// TIA Portal V18 program export: 6 tag tables, 0 data types, 2 data blocks, 13 code blocks (in call order from the OBs), 43 instance data blocks

VAR_GLOBAL   // PLC tag table "Alarms"
   "Alarm Main 1/5" AT %MW600 : Word;
   "Alarm Main 2/5" AT %MW602 : Word;
   "Alarm Main 3/5" AT %MW604 : Word;
   "Alarm Main 4/5" AT %MW606 : Word;
   "Alarm Main 5/5" AT %MW608 : Word;
   "Alarm Main 6" AT %MW610 : Word;
   "Alarm Main 7" AT %MW612 : Word;
   "AL-Drive Left Slow Limit Angle" AT %M600.0 : Bool;
   "AL-Drive Left Stop Limit LS" AT %M600.1 : Bool;
   "AL-Drive Left Stop Limit Angle" AT %M600.2 : Bool;
   "AL-Drive Left Stop Limit" AT %M600.3 : Bool;
   "AL-Drive Right Slow Limit Angle" AT %M600.4 : Bool;
   "AL-Drive Right Stop Limit LS" AT %M600.5 : Bool;
   "AL-Drive Right Stop Limit Angle" AT %M600.6 : Bool;
   "AL-Drive Right Stop Limit" AT %M600.7 : Bool;
   "AL-Rotunda Left Slow Limit" AT %M601.0 : Bool;
   "AL-Rotunda Right Slow Limit" AT %M601.1 : Bool;
   "AL-Rotunda Slow Limit" AT %M601.2 : Bool;
   "AL-Rotunda Left Stop Limit LS" AT %M601.3 : Bool;
   "AL-Rotunda Left FW Stop Limit" AT %M601.4 : Bool;
   "AL-Rotunda Left BW Stop Limit" AT %M601.5 : Bool;
   "AL-Rotunda Right Stop Limit LS" AT %M601.6 : Bool;
   "AL-Rotunda Right FW Stop Limit" AT %M601.7 : Bool;
   "AL-Rotunda Right BW Stop Limit" AT %M602.0 : Bool;
   "AL-Rotunda FW Stop Limit All" AT %M602.1 : Bool;
   "AL-Rotunda BW Stop Limit All" AT %M602.2 : Bool;
   "AL-Tunnel FW Slow Limit Laser" AT %M602.3 : Bool;
   "AL-Tunnel FW Slow Limit LS" AT %M602.4 : Bool;
   "AL-Tunnel FW Slow Limit PhotoCell" AT %M602.5 : Bool;
   "AL-Tunnel FW Slow Limit UltraSonic" AT %M602.6 : Bool;
   "AL-Tunnel FW Slow Limit All" AT %M602.7 : Bool;
   "AL-Tunnel BW Slow Limit Laser" AT %M603.0 : Bool;
   "AL-Tunnel BW Slow Limit LS" AT %M603.1 : Bool;
   "AL-Tunnel BW Slow Limit All" AT %M603.2 : Bool;
   "AL-Tunnel FW Stop Limit Laser" AT %M603.3 : Bool;
   "AL-Tunnel FW Stop Limit LS" AT %M603.4 : Bool;
   "AL-Tunnel FW Stop Limit PhotoCell Left" AT %M603.5 : Bool;
   "AL-Tunnel FW Stop Limit PhotoCell Mid" AT %M603.6 : Bool;
   "AL-Tunnel FW Stop Limit PhotoCell Right" AT %M603.7 : Bool;
   "AL-Tunnel FW Stop Limit All" AT %M604.0 : Bool;
   "AL-Tunnel FW Emergency Stop Limit" AT %M604.1 : Bool;
   "AL-Tunnel BW Stop Limit Laser" AT %M604.2 : Bool;
   "AL-Tunnel BW Stop Limit LS" AT %M604.3 : Bool;
   "AL-Tunnel BW Stop Limit All" AT %M604.4 : Bool;
   "AL-Tunnel BW Emergency Stop Limit" AT %M604.5 : Bool;
   "AL-Slow Activated" AT %M604.6 : Bool;
   "AL-Drive Slow Limit All" AT %M604.7 : Bool;
   "AL-Tunnel FW Slow Limit Slope" AT %M605.0 : Bool;
   "AL-Tunnel FW Stop Limit Slope" AT %M605.1 : Bool;
   "AL-Tunnel BW Slow Limit Slope" AT %M605.2 : Bool;
   "AL-Tunnel BW Stop Limit Slope" AT %M605.3 : Bool;
   "AL-Drivers Fault, Wheel" AT %M605.4 : Bool;
   "AL-Wheel Fuse" AT %M605.5 : Bool;
   "AL-Up Stop Limit, Wire" AT %M605.6 : Bool;
   "AL-Up Stop Limit, Max Slope" AT %M605.7 : Bool;
   "AL-Up Stop Limit, BW LS" AT %M606.0 : Bool;
   "AL-Up Stop Limit, All" AT %M606.1 : Bool;
   "AL-Down Stop Limit, Wire" AT %M606.2 : Bool;
   "AL-Down Stop Limit, Object" AT %M606.3 : Bool;
   "AL-Down Stop Limit, Min Slope" AT %M606.4 : Bool;
   "AL-Down Stop Limit, FW LS" AT %M606.5 : Bool;
   "AL-Down Stop Limit, All" AT %M606.6 : Bool;
   "AL-SafetyShoe Activated" AT %M606.7 : Bool;
   "AL-SafetyShoe Cable Problem" AT %M607.0 : Bool;
   "AL-AutoLeveller Up Over Work" AT %M607.1 : Bool;
   "AL-AutoLeveller Down Over Work" AT %M607.2 : Bool;
   "AL-AutoLeveller Touch" AT %M607.3 : Bool;
   "AL-Hydraulic Motor MKS" AT %M607.4 : Bool;
   "AL-Up Button Pressed" AT %M607.5 : Bool;
   "AL-Down Button Pressed" AT %M607.6 : Bool;
   "AL-AutoLeveller Motor Fault" AT %M607.7 : Bool;
   "AL-Left Canopy Touch" AT %M608.0 : Bool;
   "AL-Right Canopy Touch" AT %M608.1 : Bool;
   "AL-Left Canopy MKS" AT %M608.2 : Bool;
   "AL-Right Canopy MKS" AT %M608.3 : Bool;
   "AL-Canopy FW Button Pressed" AT %M608.4 : Bool;
   "AL-Canopy BW Button Pressed" AT %M608.5 : Bool;
   "AL-Cab Left Stop Limit, LS" AT %M608.6 : Bool;
   "AL-Cab Left Stop Limit, Angle" AT %M608.7 : Bool;
   "AL-Cab Left Stop Limit, All" AT %M609.0 : Bool;
   "AL-Cab Right Stop Limit, LS" AT %M609.1 : Bool;
   "AL-Cab Right Stop Limit, Angle" AT %M609.2 : Bool;
   "AL-Cab Right Stop Limit, All" AT %M609.3 : Bool;
   "AL-Driver Fault, Cab" AT %M609.4 : Bool;
   "AL-Cab Motor MKS" AT %M609.5 : Bool;
   "AL-Cab Left Button Pressed" AT %M609.6 : Bool;
   "AL-Cab Right Button Pressed" AT %M609.7 : Bool;
   "AL-Cab Floor FW Button Pressed" AT %M610.0 : Bool;
   "AL-Cab Floor BW Button Pressed" AT %M610.1 : Bool;
   "AL-Cab Floor Motor Fault" AT %M610.2 : Bool;
   "AL-PBB in Off Mode" AT %M610.3 : Bool;
   "AL-PBB in Auto Mode" AT %M610.4 : Bool;
   "AL-Left Emergency Stop Pressed" AT %M610.5 : Bool;
   "AL-Right Emergency Stop Pressed" AT %M610.6 : Bool;
   "AL-CP Emergency Stop Pressed" AT %M610.7 : Bool;
   "AL-Emergency Stop Pressed" AT %M611.0 : Bool;
   "AL-ByPass Activated" AT %M611.1 : Bool;
   "AL-PBB in On Mode" AT %M611.2 : Bool;
   "AL-Main Contactor ON" AT %M611.3 : Bool;
   "AL-FAULT" AT %M611.4 : Bool;
   "AL-SafetyBarrier Activated" AT %M611.5 : Bool;
   "AL-No Electricity" AT %M611.6 : Bool;
   "AL-Service-Hose" AT %M619.0 : Bool;
   "AL-Service-GPU" AT %M619.1 : Bool;
   "AL-Service-PCA" AT %M619.2 : Bool;
   "AL-Service" AT %M619.3 : Bool;
   "AL-Drive Angle LS FW Stop" AT %M619.5 : Bool;
   "AL-Drive Angle LS BW Stop" AT %M619.4 : Bool;
   "AL-PBB HOME" AT %M619.6 : Bool;
   "AL-AutoLeveller Down" AT %M614.0 : Bool;
   "AL-AutoLeveller Up" AT %M614.1 : Bool;
END_VAR

VAR_GLOBAL   // PLC tag table "Analog_Clock"
   "Rotunda Angle input" AT %IW160 : Int;
   "Drive Angle input" AT %IW164 : Int;
   "Cabin Angle input" AT %IW166 : Int;
   "WireDraw Encoder input" AT %IW176 : Int;
   "Laser input" AT %IW162 : Int;
   "Left Driver Analog input" AT %QW160 : Int;
   "Right Driver Analog input" AT %QW162 : Int;
   "Cab Driver Analog input" AT %QW176 : Int;
   "Slow Mode input" AT %M226.1 : Bool;
   "Canopy Touch Memo" AT %M217.4 : Bool;
END_VAR

VAR_GLOBAL   // PLC tag table "HMI"
   "HMI SafetyEdge Bypass" AT %M800.0 : Bool;
   "HMI R1 - Plane Door Light" AT %M800.1 : Bool;
   "HMI R2 - Plane Door Light" AT %M800.2 : Bool;
   "HMI R3 - Drive Unit Light" AT %M800.3 : Bool;
   "HMI R4 - Cabin Front Light" AT %M800.4 : Bool;
   "HMI R6 - SafetyEdge Light" AT %M800.5 : Bool;
   "HMI - Lamp Test Button" AT %M800.6 : Bool;
   "HMI - Floor Auto Mode" AT %M800.7 : Bool;
   "HMI - AntiCrash UltraSonic ByPass" AT %M801.0 : Bool;
   "HMI - Int Light Button" AT %M801.1 : Bool;
   "HMI - Fire Siren Acitve/Passive" AT %M801.2 : Bool;
   "HMI - Auto Floor" AT %M801.3 : Bool;
END_VAR

VAR_GLOBAL   // PLC tag table "Inputs"
   "Driver Alarm Left" AT %I0.0 : Bool;
   "Driver Fault Left" AT %I0.1 : Bool;
   "Driver Alarm Right" AT %I0.2 : Bool;
   "Driver Fault Right" AT %I0.3 : Bool;
   "Cab Driver Fault" AT %I0.5 : Bool;
   "Drive LSW Stop Left" AT %I2.0 : Bool;
   "Drive LSW Stop Right" AT %I2.1 : Bool;
   SafetyEdge AT %I2.4 : Bool;
   "Em Stop Left" AT %I2.2 : Bool;
   "Em Stop Right" AT %I2.3 : Bool;
   "Canopy Touch Left" AT %I2.7 : Bool;
   "Canopy Touch Right" AT %I3.0 : Bool;
   "Bumper Touch Left" AT %I3.1 : Bool;
   "Bumper Touch Mid" AT %I3.2 : Bool;
   "Bumper Touch Right" AT %I3.3 : Bool;
   "PhotoCell for AirCraft" AT %I3.4 : Bool;
   "UltraSonic for AirCraft" AT %I3.5 : Bool;
   "UltraSonic for Object" AT %I3.6 : Bool;
   "AutoLeveller Touch" AT %I3.7 : Bool;
   "AutoLeveller Up Sensor" AT %I4.0 : Bool;
   "AutoLeveller Down Sensor" AT %I4.1 : Bool;
   "Cabin LSW Left" AT %I4.4 : Bool;
   "Cabin LSW Right" AT %I4.5 : Bool;
   "PCA Active" AT %I15.5 : Bool;
   "Rotunda LSW Left Stop" AT %I4.6 : Bool;
   "Rotunda LSW Right Stop" AT %I4.7 : Bool;
   "Tunnel LSW FW Slow İnput" AT %I5.2 : Bool;   // FW Slow
   "Tunnel LSW BW Slow İnput" AT %I5.3 : Bool;   // BW Slow
   "Tunnel LSW FW Stop İnput" AT %I5.4 : Bool;   // FW Stop
   "Tunnel LSW BW Stop İnput" AT %I5.5 : Bool;   // BW Stop
   "Tunnel LSW FW Em Stop İnput" AT %I5.6 : Bool;   // FW Em Stop
   "Tunnel LSW BW Em Stop İnput" AT %I5.7 : Bool;   // BW Em Stop
   "Rotunda Fire Detector" AT %I6.0 : Bool;
   "Drive Wheel Fuse" AT %I6.7 : Bool;
   "Fuse Hydraulic" AT %I6.1 : Bool;
   "Fuse Cab" AT %I6.2 : Bool;
   "Phase Relay - PCR" AT %I7.0 : Bool;
   "SafetyShoe-1" AT %I10.0 : Bool;
   "SafetyShoe-2" AT %I10.1 : Bool;
   "Fuse Left Canopy" AT %I10.3 : Bool;
   "Fuse Right Canopy" AT %I10.4 : Bool;
   "Fuse Cab Floor" AT %I10.2 : Bool;
   "Fuse AutoLeveller" AT %I10.5 : Bool;
   "Button ByPass" AT %I11.0 : Bool;
   "Button Reset" AT %I11.1 : Bool;
   "Button Light Int" AT %I11.2 : Bool;
   "Button Ext Light" AT %I11.3 : Bool;
   "Button BackUp" AT %I11.4 : Bool;
   "Em Stop Button" AT %I11.5 : Bool;
   "Key-1 ON" AT %I11.7 : Bool;
   "Key-2 OFF" AT %I11.6 : Bool;
   "Cab Button Left" AT %I12.0 : Bool;
   "Cab Button Right" AT %I12.1 : Bool;
   "Button PBB Up" AT %I12.2 : Bool;
   "Button Pbb Down" AT %I12.3 : Bool;
   "Canopy Button BW" AT %I12.5 : Bool;
   "Canopy Button FW" AT %I12.4 : Bool;
   "Cab Floor FW" AT %I12.6 : Bool;
   "Cab Floor BW" AT %I12.7 : Bool;
   "JoyStick X22 L2" AT %I13.0 : Bool;
   "JoyStick X33 FW" AT %I13.1 : Bool;
   "JoyStick X44 L3" AT %I13.2 : Bool;
   "JoyStick X55 BW" AT %I13.3 : Bool;
   "JoyStick Y22 L2" AT %I13.4 : Bool;
   "JoyStick Y33 RGHT" AT %I13.5 : Bool;
   "JoyStick Y44 L3" AT %I13.6 : Bool;
   "JoyStick Y55 LFT" AT %I13.7 : Bool;
   "JoyStick 91 Brake" AT %I14.0 : Bool;
   "Fuse 1Power Supply" AT %I6.3 : Bool;
   "Fuse 2Power Supply" AT %I6.4 : Bool;
   "Fuse Phase Control Relay" AT %I6.5 : Bool;
   "GPU2 Active" AT %I15.3 : Bool;
   "Fire Detector Cabin" AT %I4.3 : Bool;
   "Fuse Hose Ritriver" AT %I6.6 : Bool;
   Fuse AT %I7.5 : Bool;
   "PCA Error" AT %I15.6 : Bool;
   "GPU2 Error" AT %I15.4 : Bool;
   "GPU1 Active" AT %I15.1 : Bool;
   "GPU1 Error" AT %I15.2 : Bool;
   "Hose Active" AT %I15.7 : Bool;
END_VAR

VAR_GLOBAL   // PLC tag table "MemoryType"
   "PBB Off Mode" AT %M200.0 : Bool;
   "PBB On Mode" AT %M200.1 : Bool;
   "PBB Auto Mode" AT %M200.2 : Bool;
   "Emergency Stop Button Pressed" AT %M200.3 : Bool;
   "Tunnel FW Em Stop LS M" AT %M200.4 : Bool;
   "Tunnel BW Em Stop LS M" AT %M200.5 : Bool;
   "Start M" AT %M200.6 : Bool;
   "Fuse Problem Major" AT %M200.7 : Bool;
   "AutoLeveller Fault" AT %M201.0 : Bool;
   "AutoLeveller Up Over Work" AT %M201.1 : Bool;
   "AutoLeveller Down Over Work" AT %M201.2 : Bool;
   "Driver Error Left" AT %M201.3 : Bool;
   "Driver Error Right" AT %M201.4 : Bool;
   "Wheel Drivers Fault" AT %M201.5 : Bool;
   "SafetyShoe Siren&Info" AT %M201.6 : Bool;
   "SafetyBarrier Activated" AT %M201.7 : Bool;
   "Fault Occurred Major" AT %M202.1 : Bool;
   "Cabin Motor Driver Fault" AT %M202.2 : Bool;
   "Fault Occured Minor" AT %M202.3 : Bool;
   OK AT %M202.4 : Bool;
   "FW L1" AT %M202.5 : Bool;
   "FW L2" AT %M202.6 : Bool;
   "FW L3" AT %M202.7 : Bool;
   "BW L1" AT %M203.0 : Bool;
   "BW L2" AT %M203.1 : Bool;
   "BW L3" AT %M203.2 : Bool;
   "LFT L1" AT %M203.3 : Bool;
   "LFT L2" AT %M203.4 : Bool;
   "LFT L3" AT %M203.5 : Bool;
   "RGHT L1" AT %M203.6 : Bool;
   "RGHT L2" AT %M203.7 : Bool;
   "RGHT L3" AT %M204.0 : Bool;
   "JS Mid M" AT %M204.1 : Bool;
   "SafetyShoe Activated" AT %M204.2 : Bool;
   "AutoLeveller Up" AT %M204.3 : Bool;
   "AutoLeveller Down" AT %M204.4 : Bool;
   "sanal kesici (1)" AT %M204.5 : Bool;
   "Down Stop Object Limit" AT %M204.6 : Bool;
   "SafetyShoe Long Press" AT %M204.7 : Bool;
   "SS Cable Problem" AT %M205.0 : Bool;
   "AutoSafety Cross" AT %M205.1 : Bool;
   "AutoLeveller FW" AT %M205.2 : Bool;
   "AutoLeveller BW" AT %M205.3 : Bool;
   "Autoleveler temp count" AT %M205.4 : Bool;
   "Fuse Problem Minor" AT %M205.7 : Bool;
   "Wire Up Stop PBB" AT %M206.0 : Bool;
   "Slope Stop Up" AT %M206.1 : Bool;
   "Wire Up Stop PBB Limit All" AT %M206.2 : Bool;
   "Wire Down Stop PBB" AT %M206.3 : Bool;
   "Slope Stop Down" AT %M206.4 : Bool;
   "Down Stop Object" AT %M206.5 : Bool;
   "Down Stop PBB All" AT %M206.6 : Bool;
   "Speed L1" AT %IW100 : Int;
   "Speed L2" AT %IW102 : Int;
   "Speed L3" AT %IW104 : Int;
   "Slow Activated" AT %M207.2 : Bool;
   "Drive Slow Limit All" AT %M207.3 : Bool;
   "FW Slow Limit All" AT %M207.4 : Bool;
   "BW Slow Limit All" AT %M207.5 : Bool;
   "FW M" AT %M207.6 : Bool;
   "BW M" AT %M207.7 : Bool;
   "FW-LFT" AT %M208.0 : Bool;
   "FW-RGHT" AT %M208.1 : Bool;
   "BW-LFT" AT %M208.2 : Bool;
   "BW-RGHT" AT %M208.3 : Bool;
   "Cross M" AT %M208.4 : Bool;
   "FW Stop All" AT %M208.5 : Bool;
   "BW Stop All" AT %M208.6 : Bool;
   "LFT Stop All" AT %M208.7 : Bool;
   "RGHT Stop All" AT %M209.0 : Bool;
   "FW Allowed" AT %M209.1 : Bool;
   "BW Allowed" AT %M209.2 : Bool;
   "LFT Allowed" AT %M209.3 : Bool;
   "RGHT Allowed" AT %M209.4 : Bool;
   "FW-LFT Allowed" AT %M209.5 : Bool;
   "FW-RGHT Allowed" AT %M209.6 : Bool;
   "BW-LFT Allowed" AT %M209.7 : Bool;
   "BW-RGHT Allowed" AT %M210.0 : Bool;
   "Drive Angle Stop Left" AT %M210.1 : Bool;
   "Drive LSW Left Stop" AT %M210.2 : Bool;
   "Drive Angle Stop Right" AT %M210.3 : Bool;
   "Drive LSW Right Stop" AT %M210.4 : Bool;
   "Drive Slow Left Limit" AT %M210.5 : Bool;
   "Drive Slow Right Limit" AT %M210.6 : Bool;
   "Rotunda FW Stop LFT" AT %M210.7 : Bool;
   "Brake Off Time" AT %ID106 : Time;
   "Rotunda BW Stop LFT" AT %M211.0 : Bool;
   "Rotunda FW Stop RGHT" AT %M211.1 : Bool;
   "Rotunda BW Stop RGHT" AT %M211.2 : Bool;
   "Rotunda FW Stop All" AT %M211.3 : Bool;
   "Rotunda BW Stop All" AT %M211.4 : Bool;
   "Tunnel Laser FW Slow Limit" AT %M211.5 : Bool;
   "Tunnel LSW FW Slow" AT %M211.6 : Bool;
   "PhotoCell Slow Limit" AT %M211.7 : Bool;
   "UltraSonic Slow Limit" AT %M212.0 : Bool;
   "AirCraft Seen Anime" AT %M212.1 : Bool;
   "Laser BW Slow Limit" AT %M212.2 : Bool;
   "LS BW Slow Limit" AT %M212.3 : Bool;
   "Laser FW Stop Limit" AT %M212.5 : Bool;
   "LS FW Stop Limit" AT %M212.7 : Bool;
   "Touch LFT Stop Limit" AT %M213.0 : Bool;
   "Touch Mid Stop Limit" AT %M213.1 : Bool;
   "Touch RGTH Stop Limit" AT %M213.2 : Bool;
   "AirCraft Touch Anime" AT %M213.3 : Bool;
   "Laser BW Stop Limit" AT %M213.4 : Bool;
   "LS BW Stop Limit" AT %M213.5 : Bool;
   "FW G120C Stop" AT %M213.7 : Bool;
   "BW G120C Stop" AT %M214.0 : Bool;
   "LFT G120C Stop" AT %M214.1 : Bool;
   "Right G120C Stop" AT %M214.2 : Bool;
   "FW-LFT G120C Stop" AT %M214.3 : Bool;
   "FW-RGHT G120C Stop" AT %M214.4 : Bool;
   "BW-LFT G120C Stop" AT %M214.5 : Bool;
   "BW-RGHT G120C Stop" AT %M214.6 : Bool;
   "Cab Angle Left Stop" AT %M214.7 : Bool;
   "Cab LS Left Stop" AT %M215.0 : Bool;
   "Cab Stop Left All" AT %M215.1 : Bool;
   "Cab Angle Right Stop" AT %M215.2 : Bool;
   "Cab LS Right Stop" AT %M215.3 : Bool;
   "Cab Stop Right All" AT %M215.4 : Bool;
   "Rotunda Stop Angle Rght" AT %M215.5 : Bool;
   "Rotunda Stop Angle LFT" AT %M215.6 : Bool;
   "Canopy BW Auto" AT %M216.0 : Bool;
   "canopy ok1" AT %M216.1 : Bool;
   "canopy ok2" AT %M216.2 : Bool;
   memo2 AT %M216.3 : Bool;
   memo AT %M216.4 : Bool;
   memo3 AT %M216.5 : Bool;
   memo4 AT %M220.0 : Bool;
   "SE ByPass" AT %M220.2 : Bool;
   "Tunnel Real Meter" AT %MD300 : Real;
   "Drive Angle Real Meter" AT %MD304 : Real;
   "Rotunda Angle Real Meter" AT %MD312 : Real;
   "Height Real" AT %MD332 : Real;
   "Cab Angle Real Meter" AT %MD348 : Real;
   "Rotunda Stop LS LFT" AT %M216.6 : Bool;
   "Rotunda Stop LS Rght" AT %M225.5 : Bool;
   "Slope Angel" AT %MD615 : Real;
   "Slope Vertical" AT %MD620 : Real;
   "Slope Stop All" AT %M225.6 : Bool;
   "Speed Active L1" AT %M225.7 : Bool;
   "Speed Active L2" AT %M226.2 : Bool;
   "Speed Active L3" AT %M226.3 : Bool;
   "Rotunda Slow Angle Rght" AT %M215.7 : Bool;
   "Rotunda Slow Angle LFT" AT %M216.7 : Bool;
   "Rotunda Slow Angle ALL" AT %M217.6 : Bool;
   "Slope Slow Down" AT %M206.7 : Bool;
   "Slope Slow Up" AT %M207.0 : Bool;
   "Slope Slow ALL" AT %M207.1 : Bool;
   "Fast Mode" AT %M226.0 : Bool;
   "Service GPU Active" AT %M202.0 : Bool;
   "Service PCA Active" AT %M205.5 : Bool;
   "Service Hose Active" AT %M205.6 : Bool;
   "Service Air Active" AT %M212.4 : Bool;
   "Drive Angle LS FW Stop" AT %M212.6 : Bool;
   "Drive Angle LS BW Stop" AT %M213.6 : Bool;
   "R6 - Cab Warning Light & Buzzer Test" AT %M226.4 : Bool;
END_VAR

VAR_GLOBAL   // PLC tag table "Outputs"
   "Left Driver On/Off" AT %Q0.0 : Bool;
   "Left Driver Reversing" AT %Q0.1 : Bool;
   "Left Driver Fault" AT %Q0.2 : Bool;
   "Left Driver DI4 STO" AT %Q0.3 : Bool;
   "Left Driver DI5 STO" AT %Q0.4 : Bool;
   "Right Driver On/Off" AT %Q0.5 : Bool;
   "Right Driver Reversing" AT %Q0.6 : Bool;
   "Right Driver Fault" AT %Q0.7 : Bool;
   "Right Driver DI4 STO" AT %Q1.0 : Bool;
   "Right Driver DI5 STO" AT %Q1.1 : Bool;
   "Cab Driver On/Off" AT %Q2.0 : Bool;
   "Cab Driver Reversing" AT %Q2.1 : Bool;
   "Cab Driver Fault Reset" AT %Q2.2 : Bool;
   "Cab Driver DI4 STO" AT %Q2.3 : Bool;
   "Cab Driver DI5 STO" AT %Q2.4 : Bool;
   "MC - Main Contactor" AT %Q3.0 : Bool;
   "C1 - Hydraulic" AT %Q3.1 : Bool;   // MC-105, MC-106, MC-107, MC-108, Cable No:200, MKS2
   "C2 - Hose power" AT %Q3.2 : Bool;
   "C3 - Tunnel Lights" AT %Q3.3 : Bool;
   "C4 - Tunnel Lights UPS" AT %Q3.4 : Bool;
   "C5 - Ext Lighting" AT %Q3.5 : Bool;
   "R2 - Bumper Red Light iptal" AT %Q3.7 : Bool;
   "R1 - SafetyEdge Red Light" AT %Q3.6 : Bool;   // MC-256 MC-257 MC-258, Cable No:204, F11
   "R4 - Mania Lights" AT %Q4.1 : Bool;
   "R6 - Cab Warning Light & Buzzer" AT %Q4.3 : Bool;
   "R7 - Motor Brake Left" AT %Q4.4 : Bool;
   "R8 - Motor Brake Right" AT %Q4.5 : Bool;
   "R12 - Valve Up" AT %Q5.1 : Bool;
   "R13 - Valve Down" AT %Q5.2 : Bool;
   "R14 - Valve Em Down" AT %Q5.3 : Bool;
   "R15 - Valve V4 & V5 Columns Down" AT %Q5.4 : Bool;
   "R3 - Left & Right Warning Lights" AT %Q4.0 : Bool;
   "R9 - Cabin Motor Brake" AT %Q4.6 : Bool;
   "R20 - PBB On" AT %Q5.5 : Bool;
   "R21 - PBB Error/Fault/Alarm" AT %Q5.6 : Bool;
   "R22 - Autoleveller On" AT %Q5.7 : Bool;
   "R23 - AutoLeveller Fault" AT %Q6.0 : Bool;
   "R24 - SafetyShoe Activated" AT %Q6.1 : Bool;
   "R25 - Fire Detector" AT %Q6.2 : Bool;
   "R50 - HMI Power" AT %Q10.0 : Bool;
   "R51 - SafetyShoe Power" AT %Q10.1 : Bool;
   "C52 - Left Canopy FW" AT %Q10.6 : Bool;
   "C53 - Left Canopy BW" AT %Q10.7 : Bool;
   "C54 - Right Canopy FW" AT %Q11.0 : Bool;
   "C55 - Right Canopy BW" AT %Q11.1 : Bool;
   "C50 - Cab Floor FW" AT %Q10.4 : Bool;
   "C51 - Cab Floor BW" AT %Q10.5 : Bool;
   "C56 - AutoLeveller FW" AT %Q11.2 : Bool;
   "C57 - AutoLeveller BW" AT %Q11.3 : Bool;
   "CP - Buzzer" AT %Q12.0 : Bool;
   "CP - Alarm Red Light" AT %Q12.1 : Bool;
   "CP - PBB Start Green Light" AT %Q12.2 : Bool;
   "CP - Reset Red Light" AT %Q12.3 : Bool;
   "CP - Button Int Lighting Light" AT %Q12.4 : Bool;
   "CP - Button Ext Lighting Light" AT %Q12.5 : Bool;
   "CP - Button Em Stop Light" AT %Q12.7 : Bool;
   "PCA Active OUT" AT %Q13.2 : Bool;
   "GPU1 Active OUT" AT %Q13.3 : Bool;
   "GPU2 Active OUT" AT %Q13.4 : Bool;
   "PBB HOME" AT %Q13.0 : Bool;
   "PBB Autoleveler ON" AT %Q13.1 : Bool;
END_VAR

DATA_BLOCK "PAutoPrePos"   // DB40
{ S7_Optimized_Access := 'TRUE' }
VERSION : 0.1
// stored: AutoNumber true, IsOnlyStoredInLoadMemory false, IsRetainMemResEnabled false, IsWriteProtectedInAS false, MemoryReserve 100
   VAR RETAIN
      "Boing 737_PBB" : Array[0..1] of Real;
      "Boing 737-Max_PBB" : Array[0..1] of Real;
      "MD 80 & 90 Series" : Array[0..1] of Real;
      "Airbus A318/319/320" : Array[0..1] of Real;
      Embraer : Array[0..1] of Real;
      "Airbus A300/310/330/340" : Array[0..1] of Real;
      "Airbus A350" : Array[0..1] of Real;
      "Boing 747/777" : Array[0..1] of Real;
   END_VAR
BEGIN
   "Boing 737_PBB"[0] := 2.77;
   "Boing 737_PBB"[1] := 40.0;
   "Boing 737-Max_PBB"[0] := 3.07;
   "Boing 737-Max_PBB"[1] := 22.0;
   "MD 80 & 90 Series"[0] := 2.4;
   "MD 80 & 90 Series"[1] := 30.0;
   "Airbus A318/319/320"[0] := 3.48;
   "Airbus A318/319/320"[1] := 48.0;
   Embraer[0] := 2.75;
   Embraer[1] := 51.0;
   "Airbus A300/310/330/340"[0] := 4.76;
   "Airbus A300/310/330/340"[1] := 35.0;
   "Airbus A350"[0] := 5.0;
   "Airbus A350"[1] := 22.0;
   "Boing 747/777"[0] := 5.0;
   "Boing 747/777"[1] := 26.0;
END_DATA_BLOCK

DATA_BLOCK "Parameters"   // DB1
{ S7_Optimized_Access := 'FALSE' }
VERSION : 0.1
// stored: AutoNumber true, IsOnlyStoredInLoadMemory false, IsWriteProtectedInAS false
   VAR RETAIN
      "Brakes On Time" : Time := T#500MS;
      "Brakes Off Time in Slow Mode" : Time := T#1S;
      "Brakes Off Time in Slow" : Time := T#200MS;
      "Brakes Off Time in Normal" : Time := T#800MS;
      "Cabin Driver Speed" : Int := 15000;
      "Canopy Up Timer" : Time := T#28S;
      "Cabin Motor Brake TOF" : Time := T#100MS;
      "Cab Angle Min" : Int := 7400;   // PBB1: -770, 19518, 0, 90, 0, 120 en sol
      "Cab Angle Max" : Int := 16500;
      "Cab Angle Min deg" : Real := 0.0;
      "Cab Angle Max deg" : Real := 135.0;
      "Cabin Stop Point Left" : Real := 0.1;
      "Cabin Stop Point Right" : Real := 135.0;
      "Drive Angle NomScale_test" : Real := 0.5;   // Ekrana sabit açı vermesi için. Test amaçlı
      "Drive Angle Min" : Int := 11750;
      "Drive Angle Max" : Int := 24000;
      "Drive Angle Min deg" : Real := 0.0;
      "Drive Angle Max deg" : Real := 180.0;
      "Drive Stop Point Left" : Real := 2.0;
      "Drive Stop Point Right" : Real := 178.0;
      "Drive Unit Stop-Slow Dif" : Real := 4.5;
      "Inclanation Desire Floor Point" : Real := 0.0;
      "Inclanation Auto Floor +- Tolerance" : Real := 0.0;
      "Laser Scale Min" : Int := 1000;
      "Laser Scale Max" : Int := 18000;
      "Laser Scale Min m" : Real := 23.5;
      "Laser Scale Max m" : Real := 36.2;
      "Laser FW Slow Point" : Real := 34.0;
      "Laser BW Slow Point" : Real := 25.0;
      "Laser FW Stop Point" : Real := 36.0;
      "Laser BW Stop Point" : Real := 23.5;
      "Laser FW Em Stop Point" : Real := 36.5;   // IPTAL
      "Laser BW Em Stop Point" : Real := 23.0;   // IPTAL
      "AutoLeveler Over Up Time" : Time := T#6S;
      "AutoLeveler Over Down Time" : Time := T#3S_500MS;
      "PBB Column Length" : Real := 5.67;
      "PBB Stop Point Up" : Real := 5.1;
      "PBB Stop Point Down" : Real := 1.8;
      "Rot Angle Min" : Int := 19850;
      "Rot Angle Max" : Int := 25850;
      "Rot Angle Min deg" : Real := 0.0;
      "Rot Angle Max deg" : Real := 180.0;
      "Rotunda Slow Point Right" : Real := 130.0;
      "Rotunda Slow Point LFT" : Real := 2.0;
      "Rotunda Stop Point Right" : Real := 135.0;
      "Rotunda Stop Point Left" : Real := 1.0;
      "Static_1 Time" : Time := T#0MS;
      "SafetyShoe Work Time" : Time := T#1S_500MS;
      "Slope Angle Min" : Real := 0.01;
      "Slope Angle Max" : Real := 7.5;
      "Slope Height Min" : Int := 0;   // PBB6:20625
      "Slope Height Max" : Int := 0;   // PBB6:17150
      "Slope Height Min m" : Real := 0.0;   // PBB6:1.57
      "Slope Height Max m" : Real := 0.0;   // PBB6:2.9
      "Slope Stop Point Max" : Real := 6.45;
      "Slope Stop Point Min" : Real := 0.1;
      "Slope Slow Point Max" : Real := 5.5;
      "Slope Slow Point Min" : Real := 0.05;
      "Speed Level 4" : Int := 4000;
      "Speed Level 1" : Int := 4000;
      "Speed Level 2" : Int := 8000;
      "Speed Level 3" : Int := 10000;
      "Wire Draw Min" : Int := 605;
      "Wire Draw Max" : Int := 15500;
      "Wire Draw Min M" : Real := 1.8;
      "Wire Draw Max M" : Real := 5.1;
      HmiDAY : Int := 29;
      HMI_MONTH : Int := 11;
      HMI_YEAR : Int := 2024;
      HMI_HOUR : Int := 15;
      HMI_MINUTE : Int := 7;
      "PLC_DAY_Set Point" : DTL := DTL#2024-08-05-00:00:00;
      HMI_DAY : DTL := DTL#2024-11-29-00:00:00;
      PLC_DAY_STOP : Bool := FALSE;
      "HMI Work Off Time" : Time := T#20M;
      "PBB Home position" : Real := 25.0;
   END_VAR
BEGIN
END_DATA_BLOCK

ORGANIZATION_BLOCK "10-Main"   // OB1, LAD, ProgramCycle
TITLE = "Main Program / "Main Program Sweep (Cycle)"
{ S7_Optimized_Access := 'TRUE' }
VERSION : 0.1
// stored: AutoNumber true, IsIECCheckEnabled false, SetENOAutomatically false
   VAR_INPUT
      Initial_Call : Bool;   // Initial call of this OB
      Remanence : Bool;   // =True, if remanent data are available
   END_VAR
   VAR_TEMP
      "Temp NormScale" : Real;
      Temp_1 : Bool;
      Temp_2 : Bool;
      "read date val" : DTL;
      "read date out" : Int;
   END_VAR
BEGIN

REGION Network 1: Off, On, Auto Definition
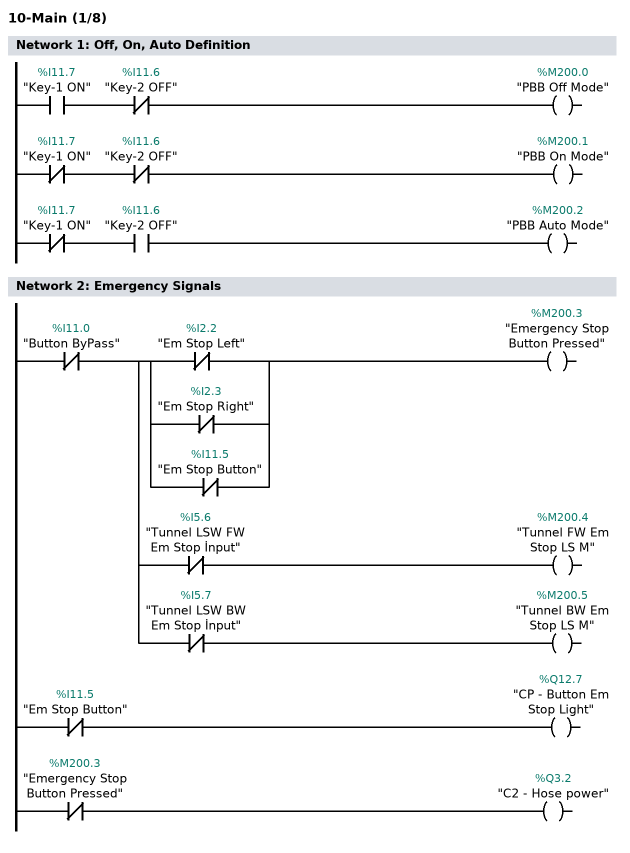
   RUNG wire#powerrail
      Contact( "Key-1 ON" )
      I_Contact( "Key-2 OFF" )
      Coil( "PBB Off Mode" )
   END_RUNG
   RUNG wire#powerrail
      I_Contact( "Key-1 ON" )
      I_Contact( "Key-2 OFF" )
      Coil( "PBB On Mode" )
   END_RUNG
   RUNG wire#powerrail
      I_Contact( "Key-1 ON" )
      Contact( "Key-2 OFF" )
      Coil( "PBB Auto Mode" )
   END_RUNG
   // the same network as SCL:
   "PBB Off Mode" := "Key-1 ON" AND NOT "Key-2 OFF";
   "PBB On Mode" := NOT "Key-1 ON" AND NOT "Key-2 OFF";
   "PBB Auto Mode" := NOT "Key-1 ON" AND "Key-2 OFF";
END_REGION

REGION Network 2: Emergency Signals
   RUNG wire#powerrail
      I_Contact( "Button ByPass" )
      wire#w1
      I_Contact( "Em Stop Left" )
      wire#w2
      Coil( "Emergency Stop Button Pressed" )
   END_RUNG
   RUNG wire#w1
      I_Contact( "Em Stop Right" )
   END_RUNG wire#w2
   RUNG wire#w1
      I_Contact( "Em Stop Button" )
   END_RUNG wire#w2
   RUNG wire#w1
      I_Contact( "Tunnel LSW FW Em Stop İnput" )
      Coil( "Tunnel FW Em Stop LS M" )
   END_RUNG
   RUNG wire#w1
      I_Contact( "Tunnel LSW BW Em Stop İnput" )
      Coil( "Tunnel BW Em Stop LS M" )
   END_RUNG
   RUNG wire#powerrail
      I_Contact( "Em Stop Button" )
      Coil( "CP - Button Em Stop Light" )
   END_RUNG
   RUNG wire#powerrail
      I_Contact( "Emergency Stop Button Pressed" )
      Coil( "C2 - Hose power" )
   END_RUNG
   // the same network as SCL:
   "Emergency Stop Button Pressed" := NOT "Button ByPass" AND (NOT "Em Stop Left" OR NOT "Em Stop Right" OR NOT "Em Stop Button");
   "Tunnel FW Em Stop LS M" := NOT "Button ByPass" AND NOT "Tunnel LSW FW Em Stop İnput";
   "Tunnel BW Em Stop LS M" := NOT "Button ByPass" AND NOT "Tunnel LSW BW Em Stop İnput";
   "CP - Button Em Stop Light" := NOT "Em Stop Button";
   "C2 - Hose power" := NOT "Emergency Stop Button Pressed";
END_REGION

REGION Network 3: Start
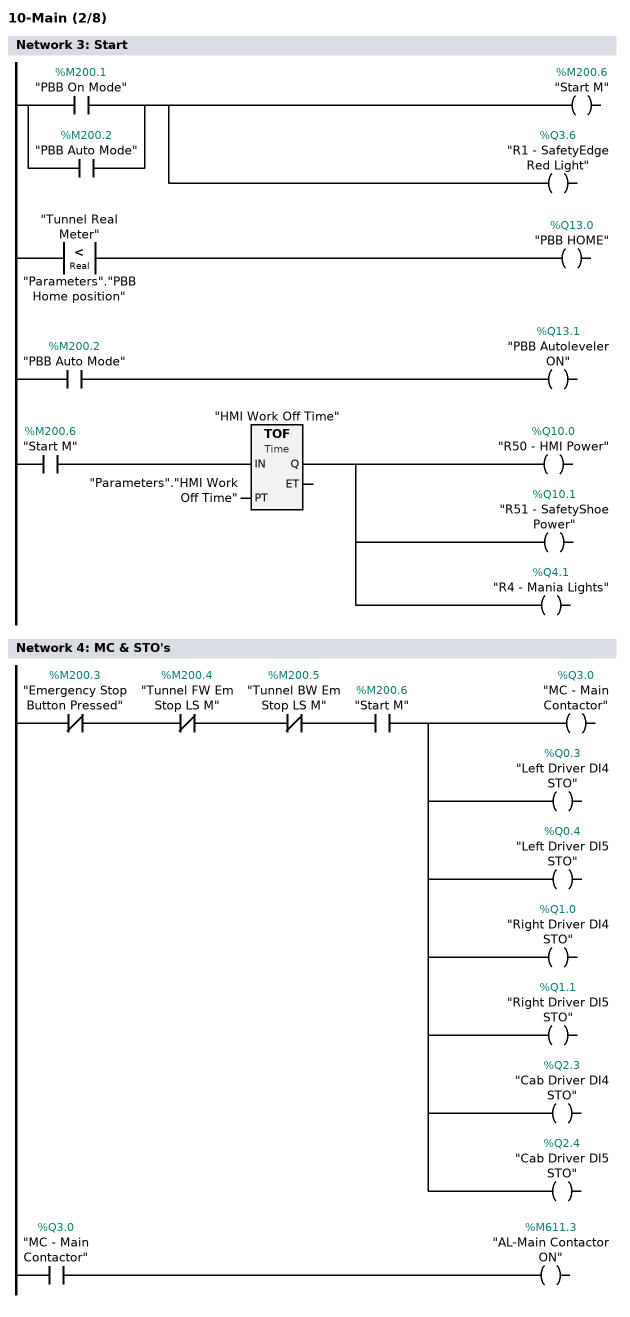
   RUNG wire#powerrail
      Contact( "PBB On Mode" )
      wire#w1
      Coil( "Start M" )
   END_RUNG
   RUNG wire#powerrail
      Contact( "PBB Auto Mode" )
   END_RUNG wire#w1
   RUNG wire#w1
      Coil( "R1 - SafetyEdge Red Light" )
   END_RUNG
   RUNG wire#powerrail
      { S7_Templates := "SrcType := Real" } LT_Contact(in1 := "Tunnel Real Meter", in2 := "Parameters"."PBB Home position")
      Coil( "PBB HOME" )
   END_RUNG
   RUNG wire#powerrail
      Contact( "PBB Auto Mode" )
      Coil( "PBB Autoleveler ON" )
   END_RUNG
   RUNG wire#powerrail
      Contact( "Start M" )
      { S7_Templates := "time_type := Time" } "HMI Work Off Time".TOF(pt := "Parameters"."HMI Work Off Time", et =>)
      wire#w2
      Coil( "R50 - HMI Power" )
   END_RUNG
   RUNG wire#w2
      Coil( "R51 - SafetyShoe Power" )
   END_RUNG
   RUNG wire#w2
      Coil( "R4 - Mania Lights" )
   END_RUNG
   // the same network as SCL:
   "Start M" := "PBB On Mode" OR "PBB Auto Mode";
   "R1 - SafetyEdge Red Light" := "Start M";
   "PBB HOME" := "Tunnel Real Meter" < "Parameters"."PBB Home position";
   "PBB Autoleveler ON" := "PBB Auto Mode";
   "HMI Work Off Time".TOF(IN := "Start M", PT := "Parameters"."HMI Work Off Time");
   "R50 - HMI Power" := "HMI Work Off Time".Q;
   "R51 - SafetyShoe Power" := "HMI Work Off Time".Q;
   "R4 - Mania Lights" := "HMI Work Off Time".Q;
END_REGION

REGION Network 4: MC & STO's
   RUNG wire#powerrail
      I_Contact( "Emergency Stop Button Pressed" )
      I_Contact( "Tunnel FW Em Stop LS M" )
      I_Contact( "Tunnel BW Em Stop LS M" )
      Contact( "Start M" )
      wire#w1
      Coil( "MC - Main Contactor" )
   END_RUNG
   RUNG wire#w1
      Coil( "Left Driver DI4 STO" )
   END_RUNG
   RUNG wire#w1
      Coil( "Left Driver DI5 STO" )
   END_RUNG
   RUNG wire#w1
      Coil( "Right Driver DI4 STO" )
   END_RUNG
   RUNG wire#w1
      Coil( "Right Driver DI5 STO" )
   END_RUNG
   RUNG wire#w1
      Coil( "Cab Driver DI4 STO" )
   END_RUNG
   RUNG wire#w1
      Coil( "Cab Driver DI5 STO" )
   END_RUNG
   RUNG wire#powerrail
      Contact( "MC - Main Contactor" )
      Coil( "AL-Main Contactor ON" )
   END_RUNG
   // the same network as SCL:
   "MC - Main Contactor" := NOT "Emergency Stop Button Pressed" AND NOT "Tunnel FW Em Stop LS M" AND NOT "Tunnel BW Em Stop LS M" AND "Start M";
   "Left Driver DI4 STO" := "MC - Main Contactor";
   "Left Driver DI5 STO" := "MC - Main Contactor";
   "Right Driver DI4 STO" := "MC - Main Contactor";
   "Right Driver DI5 STO" := "MC - Main Contactor";
   "Cab Driver DI4 STO" := "MC - Main Contactor";
   "Cab Driver DI5 STO" := "MC - Main Contactor";
   "AL-Main Contactor ON" := "MC - Main Contactor";
END_REGION

REGION Network 5: Movement OK
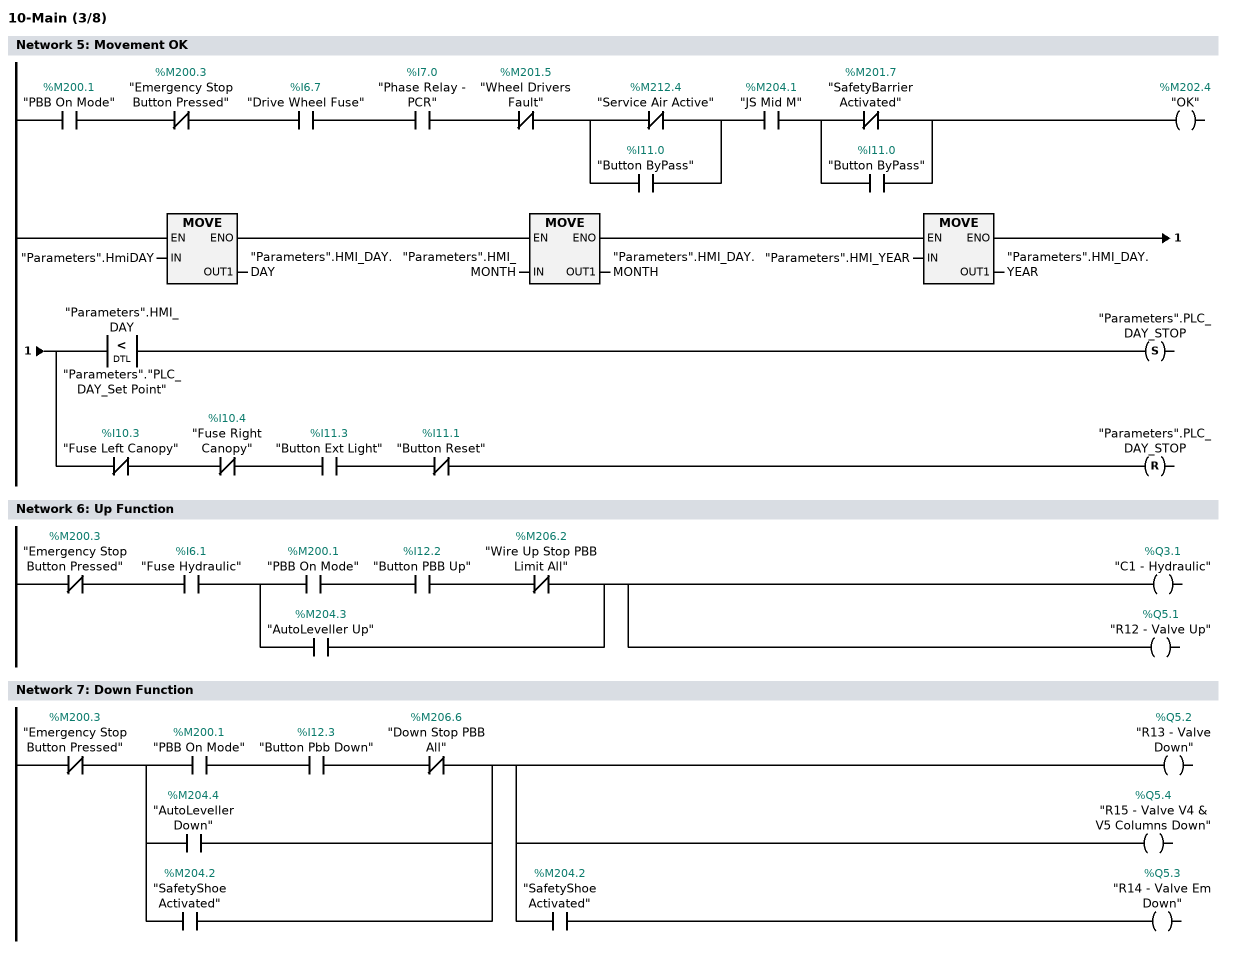
   RUNG wire#powerrail
      Contact( "PBB On Mode" )
      I_Contact( "Emergency Stop Button Pressed" )
      Contact( "Drive Wheel Fuse" )
      Contact( "Phase Relay - PCR" )
      I_Contact( "Wheel Drivers Fault" )
      wire#w1
      I_Contact( "Service Air Active" )
      wire#w2
      Contact( "JS Mid M" )
      wire#w3
      I_Contact( "SafetyBarrier Activated" )
      wire#w4
      Coil( "OK" )
   END_RUNG
   RUNG wire#w1
      Contact( "Button ByPass" )
   END_RUNG wire#w2
   RUNG wire#w3
      Contact( "Button ByPass" )
   END_RUNG wire#w4
   RUNG wire#powerrail
      Move(in := "Parameters".HmiDAY, out1 => "Parameters".HMI_DAY.DAY)
      Move(in := "Parameters".HMI_MONTH, out1 => "Parameters".HMI_DAY.MONTH)
      Move(in := "Parameters".HMI_YEAR, out1 => "Parameters".HMI_DAY.YEAR)
      wire#w5
      { S7_Templates := "SrcType := DTL" } LT_Contact(in1 := "Parameters".HMI_DAY, in2 := "Parameters"."PLC_DAY_Set Point")
      S_Coil( "Parameters".PLC_DAY_STOP )
   END_RUNG
   RUNG wire#w5
      I_Contact( "Fuse Left Canopy" )
      I_Contact( "Fuse Right Canopy" )
      Contact( "Button Ext Light" )
      I_Contact( "Button Reset" )
      R_Coil( "Parameters".PLC_DAY_STOP )
   END_RUNG
   // the same network as SCL:
   "OK" := "PBB On Mode" AND NOT "Emergency Stop Button Pressed" AND "Drive Wheel Fuse" AND "Phase Relay - PCR" AND NOT "Wheel Drivers Fault" AND (NOT "Service Air Active" OR "Button ByPass") AND "JS Mid M" AND (NOT "SafetyBarrier Activated" OR "Button ByPass");
   "Parameters".HMI_DAY.DAY := "Parameters".HmiDAY;
   "Parameters".HMI_DAY.MONTH := "Parameters".HMI_MONTH;
   "Parameters".HMI_DAY.YEAR := "Parameters".HMI_YEAR;
   IF "Parameters".HMI_DAY < "Parameters"."PLC_DAY_Set Point" THEN "Parameters".PLC_DAY_STOP := TRUE; END_IF;
   IF NOT "Fuse Left Canopy" AND NOT "Fuse Right Canopy" AND "Button Ext Light" AND NOT "Button Reset" THEN
       "Parameters".PLC_DAY_STOP := FALSE;
   END_IF;
END_REGION

REGION Network 6: Up Function
   RUNG wire#powerrail
      I_Contact( "Emergency Stop Button Pressed" )
      Contact( "Fuse Hydraulic" )
      wire#w1
      Contact( "PBB On Mode" )
      Contact( "Button PBB Up" )
      I_Contact( "Wire Up Stop PBB Limit All" )
      wire#w2
      Coil( "C1 - Hydraulic" )
   END_RUNG
   RUNG wire#w1
      Contact( "AutoLeveller Up" )
   END_RUNG wire#w2
   RUNG wire#w2
      Coil( "R12 - Valve Up" )
   END_RUNG
   // the same network as SCL:
   "C1 - Hydraulic" := NOT "Emergency Stop Button Pressed" AND "Fuse Hydraulic" AND (("PBB On Mode" AND "Button PBB Up" AND NOT "Wire Up Stop PBB Limit All") OR "AutoLeveller Up");
   "R12 - Valve Up" := "C1 - Hydraulic";
END_REGION

REGION Network 7: Down Function
   RUNG wire#powerrail
      I_Contact( "Emergency Stop Button Pressed" )
      wire#w1
      Contact( "PBB On Mode" )
      Contact( "Button Pbb Down" )
      I_Contact( "Down Stop PBB All" )
      wire#w2
      Coil( "R13 - Valve Down" )
   END_RUNG
   RUNG wire#w1
      Contact( "AutoLeveller Down" )
   END_RUNG wire#w2
   RUNG wire#w1
      Contact( "SafetyShoe Activated" )
   END_RUNG wire#w2
   RUNG wire#w2
      Coil( "R15 - Valve V4 & V5 Columns Down" )
   END_RUNG
   RUNG wire#w2
      Contact( "SafetyShoe Activated" )
      Coil( "R14 - Valve Em Down" )
   END_RUNG
   // the same network as SCL:
   "R13 - Valve Down" := NOT "Emergency Stop Button Pressed" AND (("PBB On Mode" AND "Button Pbb Down" AND NOT "Down Stop PBB All") OR "AutoLeveller Down" OR "SafetyShoe Activated");
   "R15 - Valve V4 & V5 Columns Down" := "R13 - Valve Down";
   "R14 - Valve Em Down" := "R13 - Valve Down" AND "SafetyShoe Activated";
END_REGION

REGION Network 8: Faults
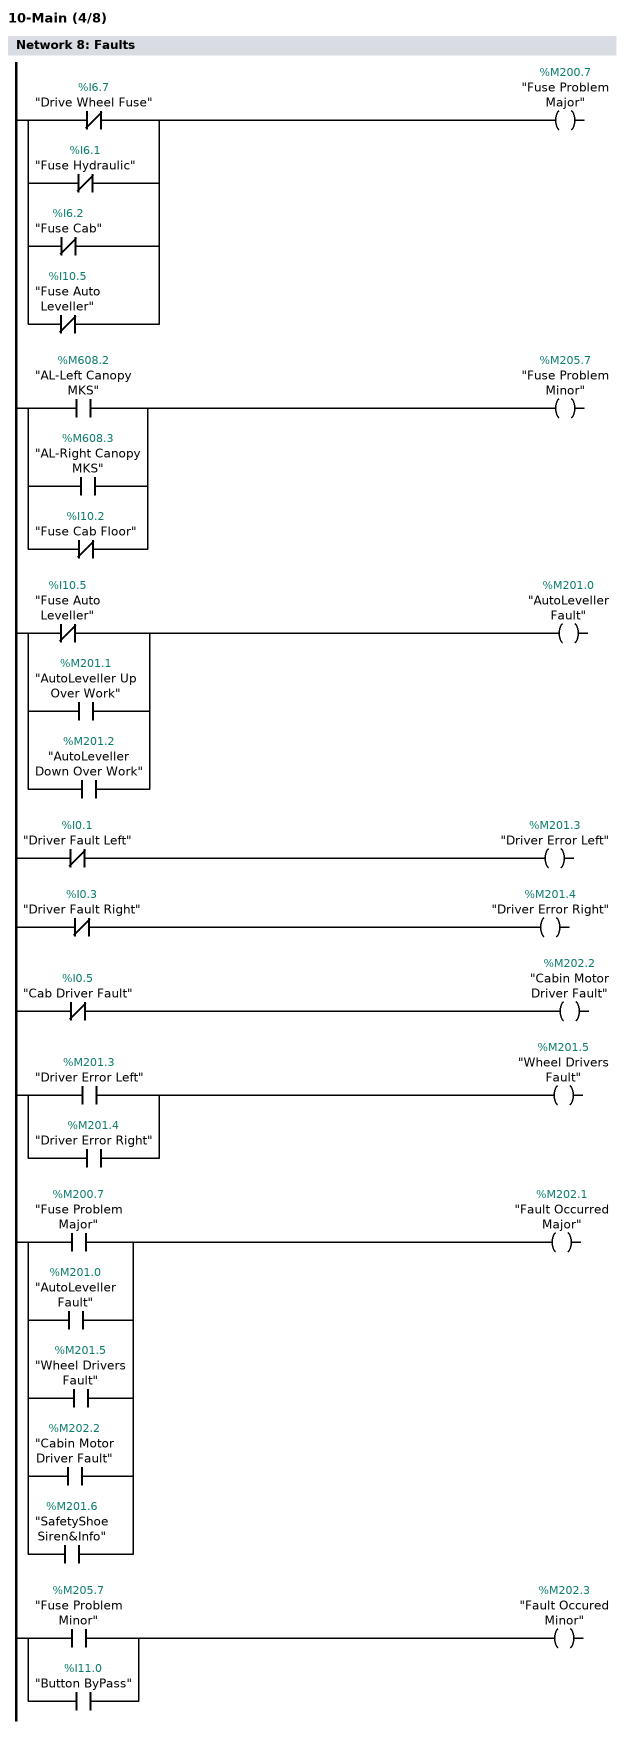
   RUNG wire#powerrail
      I_Contact( "Drive Wheel Fuse" )
      wire#w1
      Coil( "Fuse Problem Major" )
   END_RUNG
   RUNG wire#powerrail
      I_Contact( "Fuse Hydraulic" )
   END_RUNG wire#w1
   RUNG wire#powerrail
      I_Contact( "Fuse Cab" )
   END_RUNG wire#w1
   RUNG wire#powerrail
      I_Contact( "Fuse AutoLeveller" )
   END_RUNG wire#w1
   RUNG wire#powerrail
      Contact( "AL-Left Canopy MKS" )
      wire#w2
      Coil( "Fuse Problem Minor" )
   END_RUNG
   RUNG wire#powerrail
      Contact( "AL-Right Canopy MKS" )
   END_RUNG wire#w2
   RUNG wire#powerrail
      I_Contact( "Fuse Cab Floor" )
   END_RUNG wire#w2
   RUNG wire#powerrail
      I_Contact( "Fuse AutoLeveller" )
      wire#w3
      Coil( "AutoLeveller Fault" )
   END_RUNG
   RUNG wire#powerrail
      Contact( "AutoLeveller Up Over Work" )
   END_RUNG wire#w3
   RUNG wire#powerrail
      Contact( "AutoLeveller Down Over Work" )
   END_RUNG wire#w3
   RUNG wire#powerrail
      I_Contact( "Driver Fault Left" )
      Coil( "Driver Error Left" )
   END_RUNG
   RUNG wire#powerrail
      I_Contact( "Driver Fault Right" )
      Coil( "Driver Error Right" )
   END_RUNG
   RUNG wire#powerrail
      I_Contact( "Cab Driver Fault" )
      Coil( "Cabin Motor Driver Fault" )
   END_RUNG
   RUNG wire#powerrail
      Contact( "Driver Error Left" )
      wire#w4
      Coil( "Wheel Drivers Fault" )
   END_RUNG
   RUNG wire#powerrail
      Contact( "Driver Error Right" )
   END_RUNG wire#w4
   RUNG wire#powerrail
      Contact( "Fuse Problem Major" )
      wire#w5
      Coil( "Fault Occurred Major" )
   END_RUNG
   RUNG wire#powerrail
      Contact( "AutoLeveller Fault" )
   END_RUNG wire#w5
   RUNG wire#powerrail
      Contact( "Wheel Drivers Fault" )
   END_RUNG wire#w5
   RUNG wire#powerrail
      Contact( "Cabin Motor Driver Fault" )
   END_RUNG wire#w5
   RUNG wire#powerrail
      Contact( "SafetyShoe Siren&Info" )
   END_RUNG wire#w5
   RUNG wire#powerrail
      Contact( "Fuse Problem Minor" )
      wire#w6
      Coil( "Fault Occured Minor" )
   END_RUNG
   RUNG wire#powerrail
      Contact( "Button ByPass" )
   END_RUNG wire#w6
   // the same network as SCL:
   "Fuse Problem Major" := NOT "Drive Wheel Fuse" OR NOT "Fuse Hydraulic" OR NOT "Fuse Cab" OR NOT "Fuse AutoLeveller";
   "Fuse Problem Minor" := "AL-Left Canopy MKS" OR "AL-Right Canopy MKS" OR NOT "Fuse Cab Floor";
   "AutoLeveller Fault" := NOT "Fuse AutoLeveller" OR "AutoLeveller Up Over Work" OR "AutoLeveller Down Over Work";
   "Driver Error Left" := NOT "Driver Fault Left";
   "Driver Error Right" := NOT "Driver Fault Right";
   "Cabin Motor Driver Fault" := NOT "Cab Driver Fault";
   "Wheel Drivers Fault" := "Driver Error Left" OR "Driver Error Right";
   "Fault Occurred Major" := "Fuse Problem Major" OR "AutoLeveller Fault" OR "Wheel Drivers Fault" OR "Cabin Motor Driver Fault" OR "SafetyShoe Siren&Info";
   "Fault Occured Minor" := "Fuse Problem Minor" OR "Button ByPass";
END_REGION

REGION Network 9: Reset
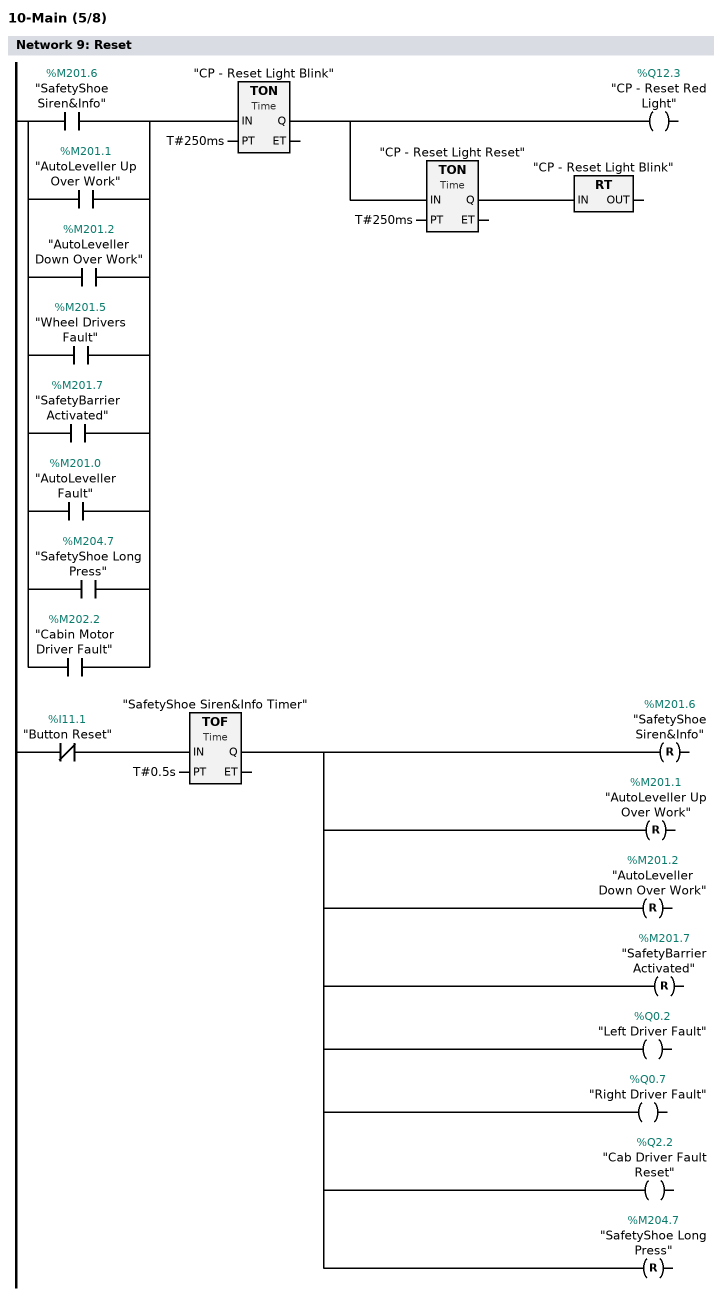
   RUNG wire#powerrail
      Contact( "SafetyShoe Siren&Info" )
      wire#w1
      { S7_Templates := "time_type := Time" } "CP - Reset Light Blink".TON(pt := T#250ms, et =>)
      wire#w2
      Coil( "CP - Reset Red Light" )
   END_RUNG
   RUNG wire#powerrail
      Contact( "AutoLeveller Up Over Work" )
   END_RUNG wire#w1
   RUNG wire#powerrail
      Contact( "AutoLeveller Down Over Work" )
   END_RUNG wire#w1
   RUNG wire#powerrail
      Contact( "Wheel Drivers Fault" )
   END_RUNG wire#w1
   RUNG wire#powerrail
      Contact( "SafetyBarrier Activated" )
   END_RUNG wire#w1
   RUNG wire#powerrail
      Contact( "AutoLeveller Fault" )
   END_RUNG wire#w1
   RUNG wire#powerrail
      Contact( "SafetyShoe Long Press" )
   END_RUNG wire#w1
   RUNG wire#powerrail
      Contact( "Cabin Motor Driver Fault" )
   END_RUNG wire#w1
   RUNG wire#w2
      { S7_Templates := "time_type := Time" } "CP - Reset Light Reset".TON(pt := T#250ms, et =>)
      RT_Coil( "CP - Reset Light Blink" )
   END_RUNG
   RUNG wire#powerrail
      I_Contact( "Button Reset" )
      { S7_Templates := "time_type := Time" } "SafetyShoe Siren&Info Timer".TOF(pt := T#0.5s, et =>)
      wire#w3
      R_Coil( "SafetyShoe Siren&Info" )
   END_RUNG
   RUNG wire#w3
      R_Coil( "AutoLeveller Up Over Work" )
   END_RUNG
   RUNG wire#w3
      R_Coil( "AutoLeveller Down Over Work" )
   END_RUNG
   RUNG wire#w3
      R_Coil( "SafetyBarrier Activated" )
   END_RUNG
   RUNG wire#w3
      Coil( "Left Driver Fault" )
   END_RUNG
   RUNG wire#w3
      Coil( "Right Driver Fault" )
   END_RUNG
   RUNG wire#w3
      Coil( "Cab Driver Fault Reset" )
   END_RUNG
   RUNG wire#w3
      R_Coil( "SafetyShoe Long Press" )
   END_RUNG
   // the same network as SCL:
   "CP - Reset Light Blink".TON(IN := "SafetyShoe Siren&Info" OR "AutoLeveller Up Over Work" OR "AutoLeveller Down Over Work" OR "Wheel Drivers Fault" OR "SafetyBarrier Activated" OR "AutoLeveller Fault" OR "SafetyShoe Long Press" OR "Cabin Motor Driver Fault",
                           PT := T#250ms);
   "CP - Reset Red Light" := "CP - Reset Light Blink".Q;
   "CP - Reset Light Reset".TON(IN := "CP - Reset Light Blink".Q, PT := T#250ms);
   IF "CP - Reset Light Reset".Q THEN RESET_TIMER("CP - Reset Light Blink"); END_IF;
   "SafetyShoe Siren&Info Timer".TOF(IN := NOT "Button Reset", PT := T#0.5s);
   IF "SafetyShoe Siren&Info Timer".Q THEN
       "SafetyShoe Siren&Info" := FALSE;
       "AutoLeveller Up Over Work" := FALSE;
       "AutoLeveller Down Over Work" := FALSE;
       "SafetyBarrier Activated" := FALSE;
   END_IF;
   "Left Driver Fault" := "SafetyShoe Siren&Info Timer".Q;
   "Right Driver Fault" := "SafetyShoe Siren&Info Timer".Q;
   "Cab Driver Fault Reset" := "SafetyShoe Siren&Info Timer".Q;
   IF "SafetyShoe Siren&Info Timer".Q THEN "SafetyShoe Long Press" := FALSE; END_IF;
END_REGION

REGION Network 10: Indicators & Warning Lights
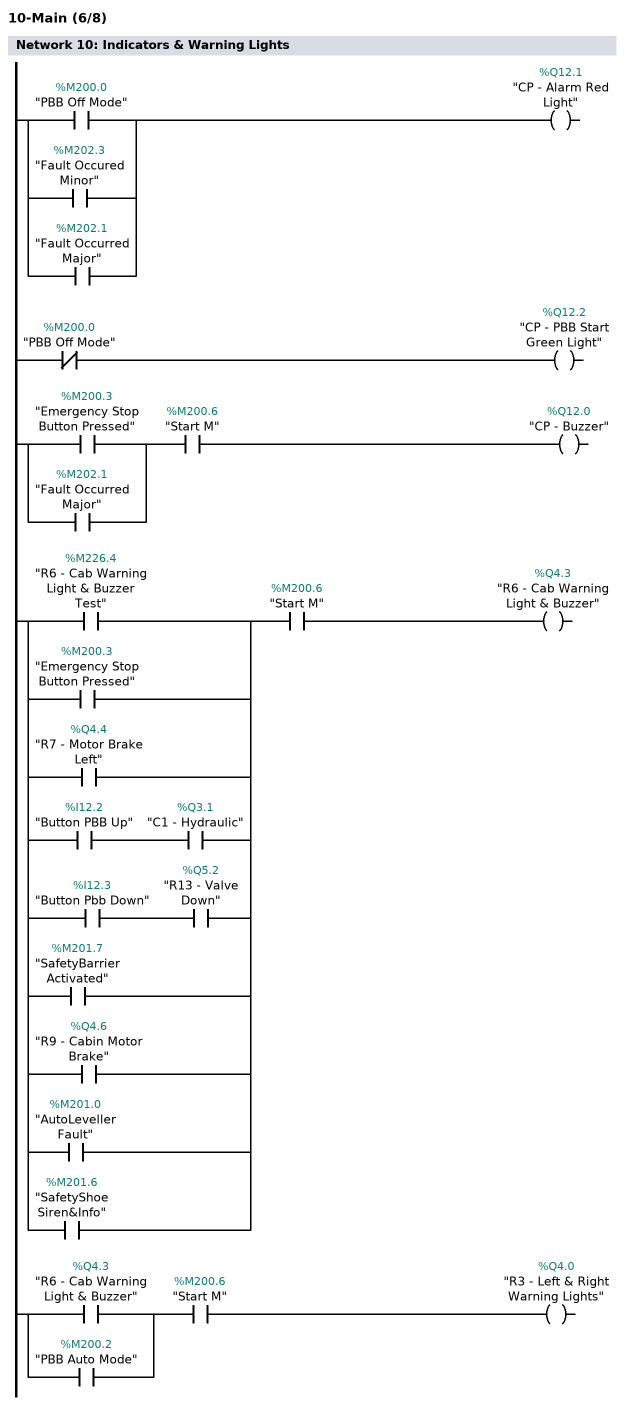
   RUNG wire#powerrail
      Contact( "PBB Off Mode" )
      wire#w1
      Coil( "CP - Alarm Red Light" )
   END_RUNG
   RUNG wire#powerrail
      Contact( "Fault Occured Minor" )
   END_RUNG wire#w1
   RUNG wire#powerrail
      Contact( "Fault Occurred Major" )
   END_RUNG wire#w1
   RUNG wire#powerrail
      I_Contact( "PBB Off Mode" )
      Coil( "CP - PBB Start Green Light" )
   END_RUNG
   RUNG wire#powerrail
      Contact( "Emergency Stop Button Pressed" )
      wire#w2
      Contact( "Start M" )
      Coil( "CP - Buzzer" )
   END_RUNG
   RUNG wire#powerrail
      Contact( "Fault Occurred Major" )
   END_RUNG wire#w2
   RUNG wire#powerrail
      Contact( "R6 - Cab Warning Light & Buzzer Test" )
      wire#w3
      Contact( "Start M" )
      Coil( "R6 - Cab Warning Light & Buzzer" )
   END_RUNG
   RUNG wire#powerrail
      Contact( "Emergency Stop Button Pressed" )
   END_RUNG wire#w3
   RUNG wire#powerrail
      Contact( "R7 - Motor Brake Left" )
   END_RUNG wire#w3
   RUNG wire#powerrail
      Contact( "Button PBB Up" )
      Contact( "C1 - Hydraulic" )
   END_RUNG wire#w3
   RUNG wire#powerrail
      Contact( "Button Pbb Down" )
      Contact( "R13 - Valve Down" )
   END_RUNG wire#w3
   RUNG wire#powerrail
      Contact( "SafetyBarrier Activated" )
   END_RUNG wire#w3
   RUNG wire#powerrail
      Contact( "R9 - Cabin Motor Brake" )
   END_RUNG wire#w3
   RUNG wire#powerrail
      Contact( "AutoLeveller Fault" )
   END_RUNG wire#w3
   RUNG wire#powerrail
      Contact( "SafetyShoe Siren&Info" )
   END_RUNG wire#w3
   RUNG wire#powerrail
      Contact( "R6 - Cab Warning Light & Buzzer" )
      wire#w4
      Contact( "Start M" )
      Coil( "R3 - Left & Right Warning Lights" )
   END_RUNG
   RUNG wire#powerrail
      Contact( "PBB Auto Mode" )
   END_RUNG wire#w4
   // the same network as SCL:
   "CP - Alarm Red Light" := "PBB Off Mode" OR "Fault Occured Minor" OR "Fault Occurred Major";
   "CP - PBB Start Green Light" := NOT "PBB Off Mode";
   "CP - Buzzer" := ("Emergency Stop Button Pressed" OR "Fault Occurred Major") AND "Start M";
   "R6 - Cab Warning Light & Buzzer" := ("R6 - Cab Warning Light & Buzzer Test" OR "Emergency Stop Button Pressed" OR "R7 - Motor Brake Left" OR ("Button PBB Up" AND "C1 - Hydraulic") OR ("Button Pbb Down" AND "R13 - Valve Down") OR "SafetyBarrier Activated" OR "R9 - Cabin Motor Brake" OR "AutoLeveller Fault" OR "SafetyShoe Siren&Info") AND "Start M";
   "R3 - Left & Right Warning Lights" := ("R6 - Cab Warning Light & Buzzer" OR "PBB Auto Mode") AND "Start M";
END_REGION

REGION Network 11: Interior Lights
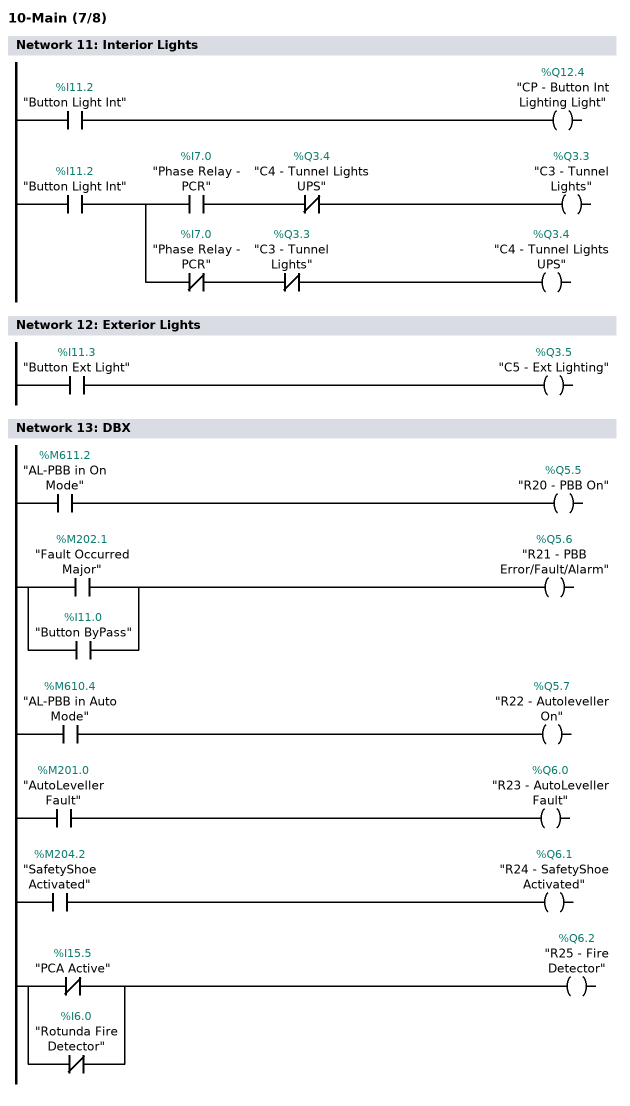
   RUNG wire#powerrail
      Contact( "Button Light Int" )
      Coil( "CP - Button Int Lighting Light" )
   END_RUNG
   RUNG wire#powerrail
      Contact( "Button Light Int" )
      wire#w1
      Contact( "Phase Relay - PCR" )
      I_Contact( "C4 - Tunnel Lights UPS" )
      Coil( "C3 - Tunnel Lights" )
   END_RUNG
   RUNG wire#w1
      I_Contact( "Phase Relay - PCR" )
      I_Contact( "C3 - Tunnel Lights" )
      Coil( "C4 - Tunnel Lights UPS" )
   END_RUNG
   // the same network as SCL:
   "CP - Button Int Lighting Light" := "Button Light Int";
   "C3 - Tunnel Lights" := "Button Light Int" AND "Phase Relay - PCR" AND NOT "C4 - Tunnel Lights UPS";
   "C4 - Tunnel Lights UPS" := "Button Light Int" AND NOT "Phase Relay - PCR" AND NOT "C3 - Tunnel Lights";
END_REGION

REGION Network 12: Exterior Lights
   RUNG wire#powerrail
      Contact( "Button Ext Light" )
      Coil( "C5 - Ext Lighting" )
   END_RUNG
   // the same network as SCL:
   "C5 - Ext Lighting" := "Button Ext Light";
END_REGION

REGION Network 13: DBX
   RUNG wire#powerrail
      Contact( "AL-PBB in On Mode" )
      Coil( "R20 - PBB On" )
   END_RUNG
   RUNG wire#powerrail
      Contact( "Fault Occurred Major" )
      wire#w1
      Coil( "R21 - PBB Error/Fault/Alarm" )
   END_RUNG
   RUNG wire#powerrail
      Contact( "Button ByPass" )
   END_RUNG wire#w1
   RUNG wire#powerrail
      Contact( "AL-PBB in Auto Mode" )
      Coil( "R22 - Autoleveller On" )
   END_RUNG
   RUNG wire#powerrail
      Contact( "AutoLeveller Fault" )
      Coil( "R23 - AutoLeveller Fault" )
   END_RUNG
   RUNG wire#powerrail
      Contact( "SafetyShoe Activated" )
      Coil( "R24 - SafetyShoe Activated" )
   END_RUNG
   RUNG wire#powerrail
      I_Contact( "PCA Active" )
      wire#w2
      Coil( "R25 - Fire Detector" )
   END_RUNG
   RUNG wire#powerrail
      I_Contact( "Rotunda Fire Detector" )
   END_RUNG wire#w2
   // the same network as SCL:
   "R20 - PBB On" := "AL-PBB in On Mode";
   "R21 - PBB Error/Fault/Alarm" := "Fault Occurred Major" OR "Button ByPass";
   "R22 - Autoleveller On" := "AL-PBB in Auto Mode";
   "R23 - AutoLeveller Fault" := "AutoLeveller Fault";
   "R24 - SafetyShoe Activated" := "SafetyShoe Activated";
   "R25 - Fire Detector" := NOT "PCA Active" OR NOT "Rotunda Fire Detector";
END_REGION

REGION Network 14: PCA and GPU Service
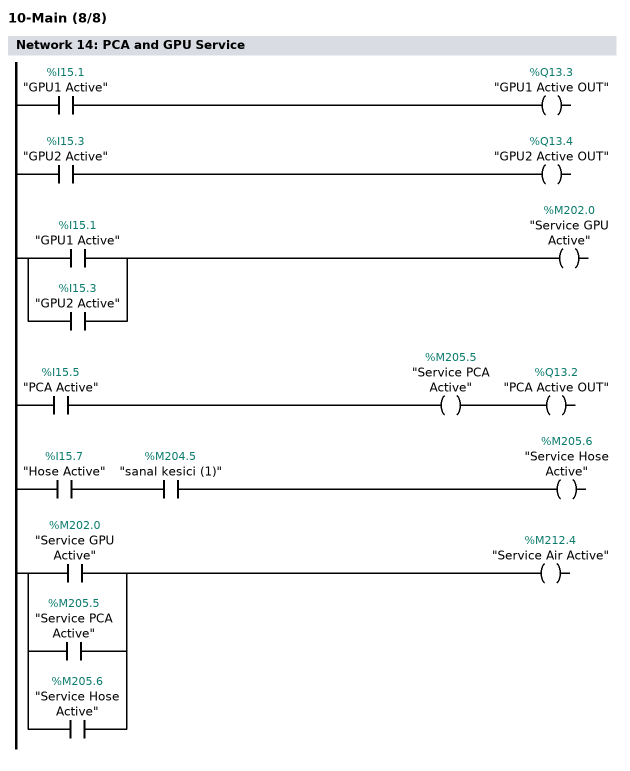
   RUNG wire#powerrail
      Contact( "GPU1 Active" )
      Coil( "GPU1 Active OUT" )
   END_RUNG
   RUNG wire#powerrail
      Contact( "GPU2 Active" )
      Coil( "GPU2 Active OUT" )
   END_RUNG
   RUNG wire#powerrail
      Contact( "GPU1 Active" )
      wire#w1
      Coil( "Service GPU Active" )
   END_RUNG
   RUNG wire#powerrail
      Contact( "GPU2 Active" )
   END_RUNG wire#w1
   RUNG wire#powerrail
      Contact( "PCA Active" )
      Coil( "Service PCA Active" )
      Coil( "PCA Active OUT" )
   END_RUNG
   RUNG wire#powerrail
      Contact( "Hose Active" )
      Contact( "sanal kesici (1)" )
      Coil( "Service Hose Active" )
   END_RUNG
   RUNG wire#powerrail
      Contact( "Service GPU Active" )
      wire#w2
      Coil( "Service Air Active" )
   END_RUNG
   RUNG wire#powerrail
      Contact( "Service PCA Active" )
   END_RUNG wire#w2
   RUNG wire#powerrail
      Contact( "Service Hose Active" )
   END_RUNG wire#w2
   // the same network as SCL:
   "GPU1 Active OUT" := "GPU1 Active";
   "GPU2 Active OUT" := "GPU2 Active";
   "Service GPU Active" := "GPU1 Active" OR "GPU2 Active";
   "Service PCA Active" := "PCA Active";
   "PCA Active OUT" := "PCA Active";
   "Service Hose Active" := "Hose Active" AND "sanal kesici (1)";
   "Service Air Active" := "Service GPU Active" OR "Service PCA Active" OR "Service Hose Active";
END_REGION
END_ORGANIZATION_BLOCK

ORGANIZATION_BLOCK "00-Alarms"   // OB126, LAD, ProgramCycle
TITLE = Alarms / "Main Program Sweep (Cycle)"
{ S7_Optimized_Access := 'TRUE' }
VERSION : 0.1
// stored: AutoNumber true, IsIECCheckEnabled false, SetENOAutomatically false
   VAR_INPUT
      Initial_Call : Bool;   // Initial call of this OB
      Remanence : Bool;   // =True, if remanent data are available
   END_VAR
BEGIN

REGION Network 1
   // Sınıflandıramadığım Alarm Listesi
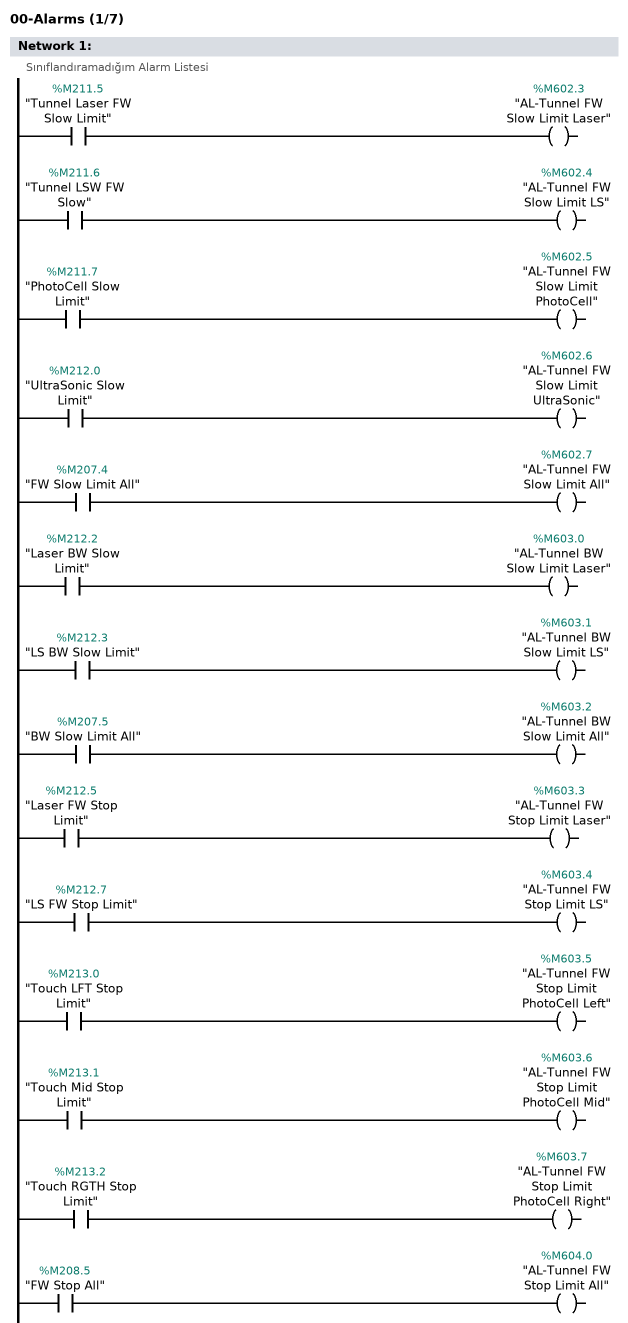
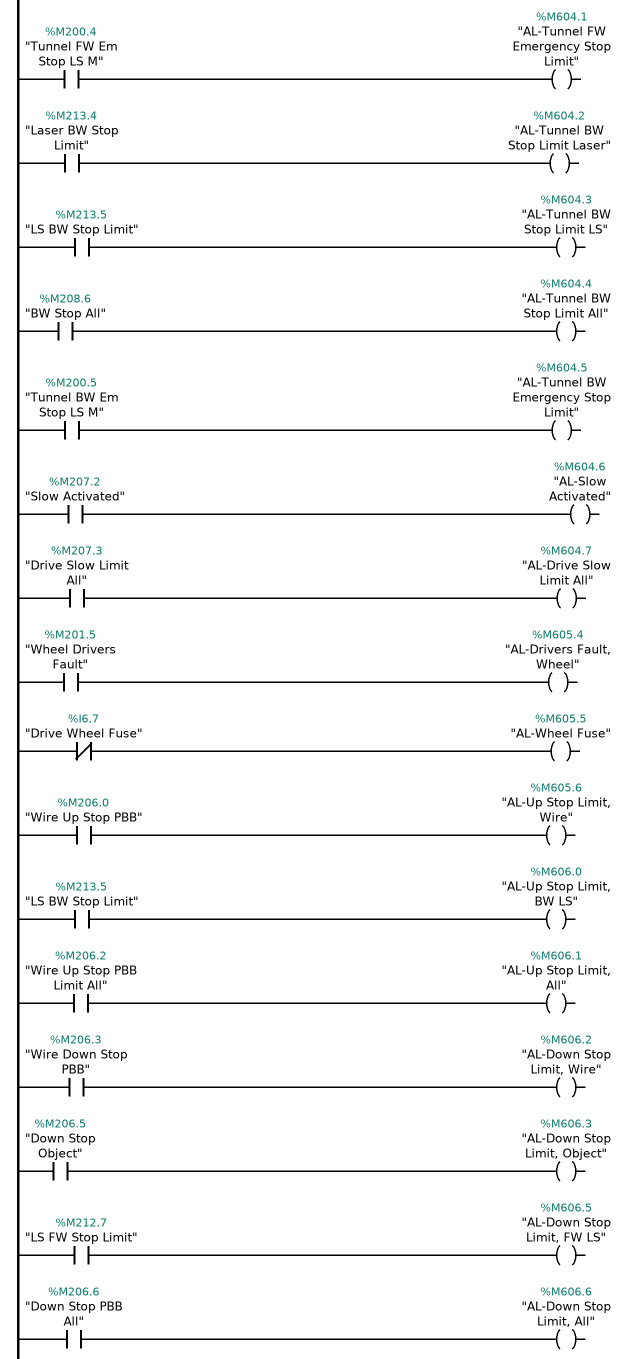
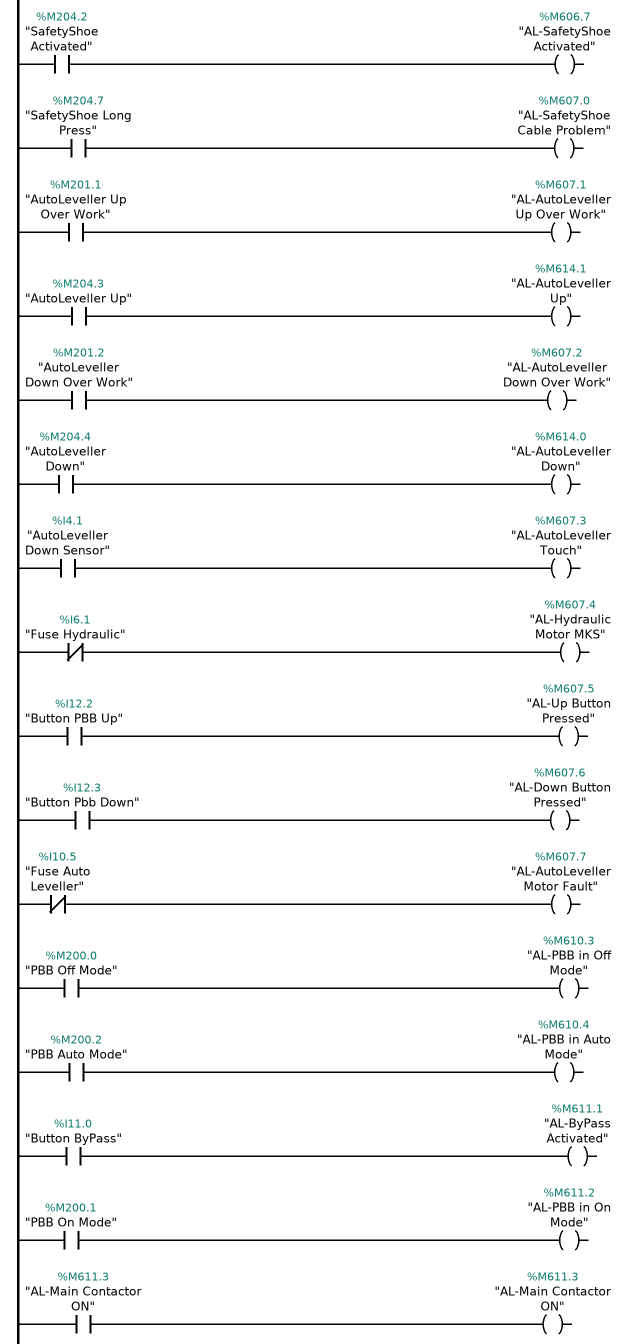
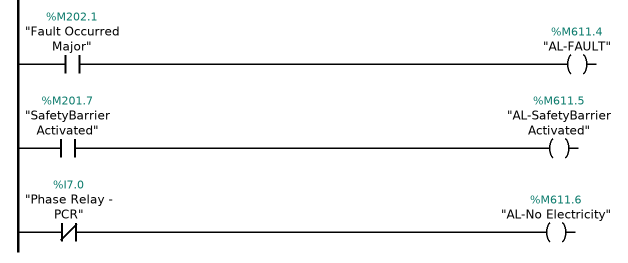
   RUNG wire#powerrail
      Contact( "Tunnel Laser FW Slow Limit" )
      Coil( "AL-Tunnel FW Slow Limit Laser" )
   END_RUNG
   RUNG wire#powerrail
      Contact( "Tunnel LSW FW Slow" )
      Coil( "AL-Tunnel FW Slow Limit LS" )
   END_RUNG
   RUNG wire#powerrail
      Contact( "PhotoCell Slow Limit" )
      Coil( "AL-Tunnel FW Slow Limit PhotoCell" )
   END_RUNG
   RUNG wire#powerrail
      Contact( "UltraSonic Slow Limit" )
      Coil( "AL-Tunnel FW Slow Limit UltraSonic" )
   END_RUNG
   RUNG wire#powerrail
      Contact( "FW Slow Limit All" )
      Coil( "AL-Tunnel FW Slow Limit All" )
   END_RUNG
   RUNG wire#powerrail
      Contact( "Laser BW Slow Limit" )
      Coil( "AL-Tunnel BW Slow Limit Laser" )
   END_RUNG
   RUNG wire#powerrail
      Contact( "LS BW Slow Limit" )
      Coil( "AL-Tunnel BW Slow Limit LS" )
   END_RUNG
   RUNG wire#powerrail
      Contact( "BW Slow Limit All" )
      Coil( "AL-Tunnel BW Slow Limit All" )
   END_RUNG
   RUNG wire#powerrail
      Contact( "Laser FW Stop Limit" )
      Coil( "AL-Tunnel FW Stop Limit Laser" )
   END_RUNG
   RUNG wire#powerrail
      Contact( "LS FW Stop Limit" )
      Coil( "AL-Tunnel FW Stop Limit LS" )
   END_RUNG
   RUNG wire#powerrail
      Contact( "Touch LFT Stop Limit" )
      Coil( "AL-Tunnel FW Stop Limit PhotoCell Left" )
   END_RUNG
   RUNG wire#powerrail
      Contact( "Touch Mid Stop Limit" )
      Coil( "AL-Tunnel FW Stop Limit PhotoCell Mid" )
   END_RUNG
   RUNG wire#powerrail
      Contact( "Touch RGTH Stop Limit" )
      Coil( "AL-Tunnel FW Stop Limit PhotoCell Right" )
   END_RUNG
   RUNG wire#powerrail
      Contact( "FW Stop All" )
      Coil( "AL-Tunnel FW Stop Limit All" )
   END_RUNG
   RUNG wire#powerrail
      Contact( "Tunnel FW Em Stop LS M" )
      Coil( "AL-Tunnel FW Emergency Stop Limit" )
   END_RUNG
   RUNG wire#powerrail
      Contact( "Laser BW Stop Limit" )
      Coil( "AL-Tunnel BW Stop Limit Laser" )
   END_RUNG
   RUNG wire#powerrail
      Contact( "LS BW Stop Limit" )
      Coil( "AL-Tunnel BW Stop Limit LS" )
   END_RUNG
   RUNG wire#powerrail
      Contact( "BW Stop All" )
      Coil( "AL-Tunnel BW Stop Limit All" )
   END_RUNG
   RUNG wire#powerrail
      Contact( "Tunnel BW Em Stop LS M" )
      Coil( "AL-Tunnel BW Emergency Stop Limit" )
   END_RUNG
   RUNG wire#powerrail
      Contact( "Slow Activated" )
      Coil( "AL-Slow Activated" )
   END_RUNG
   RUNG wire#powerrail
      Contact( "Drive Slow Limit All" )
      Coil( "AL-Drive Slow Limit All" )
   END_RUNG
   RUNG wire#powerrail
      Contact( "Wheel Drivers Fault" )
      Coil( "AL-Drivers Fault, Wheel" )
   END_RUNG
   RUNG wire#powerrail
      I_Contact( "Drive Wheel Fuse" )
      Coil( "AL-Wheel Fuse" )
   END_RUNG
   RUNG wire#powerrail
      Contact( "Wire Up Stop PBB" )
      Coil( "AL-Up Stop Limit, Wire" )
   END_RUNG
   RUNG wire#powerrail
      Contact( "LS BW Stop Limit" )
      Coil( "AL-Up Stop Limit, BW LS" )
   END_RUNG
   RUNG wire#powerrail
      Contact( "Wire Up Stop PBB Limit All" )
      Coil( "AL-Up Stop Limit, All" )
   END_RUNG
   RUNG wire#powerrail
      Contact( "Wire Down Stop PBB" )
      Coil( "AL-Down Stop Limit, Wire" )
   END_RUNG
   RUNG wire#powerrail
      Contact( "Down Stop Object" )
      Coil( "AL-Down Stop Limit, Object" )
   END_RUNG
   RUNG wire#powerrail
      Contact( "LS FW Stop Limit" )
      Coil( "AL-Down Stop Limit, FW LS" )
   END_RUNG
   RUNG wire#powerrail
      Contact( "Down Stop PBB All" )
      Coil( "AL-Down Stop Limit, All" )
   END_RUNG
   RUNG wire#powerrail
      Contact( "SafetyShoe Activated" )
      Coil( "AL-SafetyShoe Activated" )
   END_RUNG
   RUNG wire#powerrail
      Contact( "SafetyShoe Long Press" )
      Coil( "AL-SafetyShoe Cable Problem" )
   END_RUNG
   RUNG wire#powerrail
      Contact( "AutoLeveller Up Over Work" )
      Coil( "AL-AutoLeveller Up Over Work" )
   END_RUNG
   RUNG wire#powerrail
      Contact( "AutoLeveller Up" )
      Coil( "AL-AutoLeveller Up" )
   END_RUNG
   RUNG wire#powerrail
      Contact( "AutoLeveller Down Over Work" )
      Coil( "AL-AutoLeveller Down Over Work" )
   END_RUNG
   RUNG wire#powerrail
      Contact( "AutoLeveller Down" )
      Coil( "AL-AutoLeveller Down" )
   END_RUNG
   RUNG wire#powerrail
      Contact( "AutoLeveller Down Sensor" )
      Coil( "AL-AutoLeveller Touch" )
   END_RUNG
   RUNG wire#powerrail
      I_Contact( "Fuse Hydraulic" )
      Coil( "AL-Hydraulic Motor MKS" )
   END_RUNG
   RUNG wire#powerrail
      Contact( "Button PBB Up" )
      Coil( "AL-Up Button Pressed" )
   END_RUNG
   RUNG wire#powerrail
      Contact( "Button Pbb Down" )
      Coil( "AL-Down Button Pressed" )
   END_RUNG
   RUNG wire#powerrail
      I_Contact( "Fuse AutoLeveller" )
      Coil( "AL-AutoLeveller Motor Fault" )
   END_RUNG
   RUNG wire#powerrail
      Contact( "PBB Off Mode" )
      Coil( "AL-PBB in Off Mode" )
   END_RUNG
   RUNG wire#powerrail
      Contact( "PBB Auto Mode" )
      Coil( "AL-PBB in Auto Mode" )
   END_RUNG
   RUNG wire#powerrail
      Contact( "Button ByPass" )
      Coil( "AL-ByPass Activated" )
   END_RUNG
   RUNG wire#powerrail
      Contact( "PBB On Mode" )
      Coil( "AL-PBB in On Mode" )
   END_RUNG
   RUNG wire#powerrail
      Contact( "AL-Main Contactor ON" )
      Coil( "AL-Main Contactor ON" )
   END_RUNG
   RUNG wire#powerrail
      Contact( "Fault Occurred Major" )
      Coil( "AL-FAULT" )
   END_RUNG
   RUNG wire#powerrail
      Contact( "SafetyBarrier Activated" )
      Coil( "AL-SafetyBarrier Activated" )
   END_RUNG
   RUNG wire#powerrail
      I_Contact( "Phase Relay - PCR" )
      Coil( "AL-No Electricity" )
   END_RUNG
   // the same network as SCL:
   "AL-Tunnel FW Slow Limit Laser" := "Tunnel Laser FW Slow Limit";
   "AL-Tunnel FW Slow Limit LS" := "Tunnel LSW FW Slow";
   "AL-Tunnel FW Slow Limit PhotoCell" := "PhotoCell Slow Limit";
   "AL-Tunnel FW Slow Limit UltraSonic" := "UltraSonic Slow Limit";
   "AL-Tunnel FW Slow Limit All" := "FW Slow Limit All";
   "AL-Tunnel BW Slow Limit Laser" := "Laser BW Slow Limit";
   "AL-Tunnel BW Slow Limit LS" := "LS BW Slow Limit";
   "AL-Tunnel BW Slow Limit All" := "BW Slow Limit All";
   "AL-Tunnel FW Stop Limit Laser" := "Laser FW Stop Limit";
   "AL-Tunnel FW Stop Limit LS" := "LS FW Stop Limit";
   "AL-Tunnel FW Stop Limit PhotoCell Left" := "Touch LFT Stop Limit";
   "AL-Tunnel FW Stop Limit PhotoCell Mid" := "Touch Mid Stop Limit";
   "AL-Tunnel FW Stop Limit PhotoCell Right" := "Touch RGTH Stop Limit";
   "AL-Tunnel FW Stop Limit All" := "FW Stop All";
   "AL-Tunnel FW Emergency Stop Limit" := "Tunnel FW Em Stop LS M";
   "AL-Tunnel BW Stop Limit Laser" := "Laser BW Stop Limit";
   "AL-Tunnel BW Stop Limit LS" := "LS BW Stop Limit";
   "AL-Tunnel BW Stop Limit All" := "BW Stop All";
   "AL-Tunnel BW Emergency Stop Limit" := "Tunnel BW Em Stop LS M";
   "AL-Slow Activated" := "Slow Activated";
   "AL-Drive Slow Limit All" := "Drive Slow Limit All";
   "AL-Drivers Fault, Wheel" := "Wheel Drivers Fault";
   "AL-Wheel Fuse" := NOT "Drive Wheel Fuse";
   "AL-Up Stop Limit, Wire" := "Wire Up Stop PBB";
   "AL-Up Stop Limit, BW LS" := "LS BW Stop Limit";
   "AL-Up Stop Limit, All" := "Wire Up Stop PBB Limit All";
   "AL-Down Stop Limit, Wire" := "Wire Down Stop PBB";
   "AL-Down Stop Limit, Object" := "Down Stop Object";
   "AL-Down Stop Limit, FW LS" := "LS FW Stop Limit";
   "AL-Down Stop Limit, All" := "Down Stop PBB All";
   "AL-SafetyShoe Activated" := "SafetyShoe Activated";
   "AL-SafetyShoe Cable Problem" := "SafetyShoe Long Press";
   "AL-AutoLeveller Up Over Work" := "AutoLeveller Up Over Work";
   "AL-AutoLeveller Up" := "AutoLeveller Up";
   "AL-AutoLeveller Down Over Work" := "AutoLeveller Down Over Work";
   "AL-AutoLeveller Down" := "AutoLeveller Down";
   "AL-AutoLeveller Touch" := "AutoLeveller Down Sensor";
   "AL-Hydraulic Motor MKS" := NOT "Fuse Hydraulic";
   "AL-Up Button Pressed" := "Button PBB Up";
   "AL-Down Button Pressed" := "Button Pbb Down";
   "AL-AutoLeveller Motor Fault" := NOT "Fuse AutoLeveller";
   "AL-PBB in Off Mode" := "PBB Off Mode";
   "AL-PBB in Auto Mode" := "PBB Auto Mode";
   "AL-ByPass Activated" := "Button ByPass";
   "AL-PBB in On Mode" := "PBB On Mode";
   "AL-Main Contactor ON" := "AL-Main Contactor ON";
   "AL-FAULT" := "Fault Occurred Major";
   "AL-SafetyBarrier Activated" := "SafetyBarrier Activated";
   "AL-No Electricity" := NOT "Phase Relay - PCR";
END_REGION

REGION Network 2: Drive
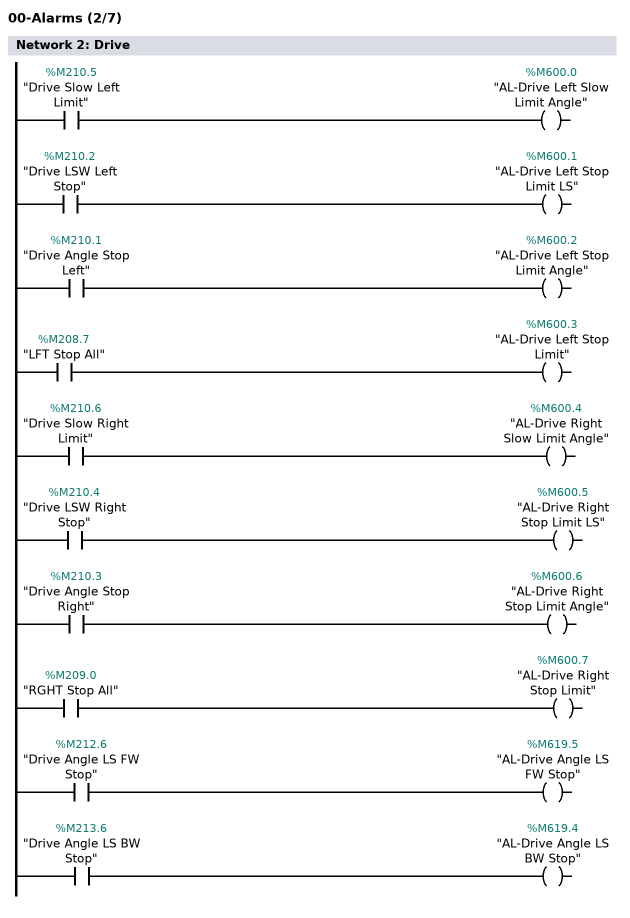
   RUNG wire#powerrail
      Contact( "Drive Slow Left Limit" )
      Coil( "AL-Drive Left Slow Limit Angle" )
   END_RUNG
   RUNG wire#powerrail
      Contact( "Drive LSW Left Stop" )
      Coil( "AL-Drive Left Stop Limit LS" )
   END_RUNG
   RUNG wire#powerrail
      Contact( "Drive Angle Stop Left" )
      Coil( "AL-Drive Left Stop Limit Angle" )
   END_RUNG
   RUNG wire#powerrail
      Contact( "LFT Stop All" )
      Coil( "AL-Drive Left Stop Limit" )
   END_RUNG
   RUNG wire#powerrail
      Contact( "Drive Slow Right Limit" )
      Coil( "AL-Drive Right Slow Limit Angle" )
   END_RUNG
   RUNG wire#powerrail
      Contact( "Drive LSW Right Stop" )
      Coil( "AL-Drive Right Stop Limit LS" )
   END_RUNG
   RUNG wire#powerrail
      Contact( "Drive Angle Stop Right" )
      Coil( "AL-Drive Right Stop Limit Angle" )
   END_RUNG
   RUNG wire#powerrail
      Contact( "RGHT Stop All" )
      Coil( "AL-Drive Right Stop Limit" )
   END_RUNG
   RUNG wire#powerrail
      Contact( "Drive Angle LS FW Stop" )
      Coil( "AL-Drive Angle LS FW Stop" )
   END_RUNG
   RUNG wire#powerrail
      Contact( "Drive Angle LS BW Stop" )
      Coil( "AL-Drive Angle LS BW Stop" )
   END_RUNG
   // the same network as SCL:
   "AL-Drive Left Slow Limit Angle" := "Drive Slow Left Limit";
   "AL-Drive Left Stop Limit LS" := "Drive LSW Left Stop";
   "AL-Drive Left Stop Limit Angle" := "Drive Angle Stop Left";
   "AL-Drive Left Stop Limit" := "LFT Stop All";
   "AL-Drive Right Slow Limit Angle" := "Drive Slow Right Limit";
   "AL-Drive Right Stop Limit LS" := "Drive LSW Right Stop";
   "AL-Drive Right Stop Limit Angle" := "Drive Angle Stop Right";
   "AL-Drive Right Stop Limit" := "RGHT Stop All";
   "AL-Drive Angle LS FW Stop" := "Drive Angle LS FW Stop";
   "AL-Drive Angle LS BW Stop" := "Drive Angle LS BW Stop";
END_REGION

REGION Network 3: Slope
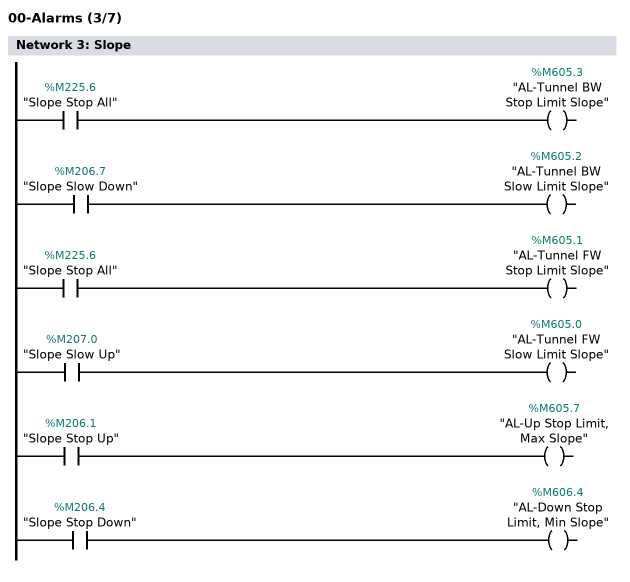
   RUNG wire#powerrail
      Contact( "Slope Stop All" )
      Coil( "AL-Tunnel BW Stop Limit Slope" )
   END_RUNG
   RUNG wire#powerrail
      Contact( "Slope Slow Down" )
      Coil( "AL-Tunnel BW Slow Limit Slope" )
   END_RUNG
   RUNG wire#powerrail
      Contact( "Slope Stop All" )
      Coil( "AL-Tunnel FW Stop Limit Slope" )
   END_RUNG
   RUNG wire#powerrail
      Contact( "Slope Slow Up" )
      Coil( "AL-Tunnel FW Slow Limit Slope" )
   END_RUNG
   RUNG wire#powerrail
      Contact( "Slope Stop Up" )
      Coil( "AL-Up Stop Limit, Max Slope" )
   END_RUNG
   RUNG wire#powerrail
      Contact( "Slope Stop Down" )
      Coil( "AL-Down Stop Limit, Min Slope" )
   END_RUNG
   // the same network as SCL:
   "AL-Tunnel BW Stop Limit Slope" := "Slope Stop All";
   "AL-Tunnel BW Slow Limit Slope" := "Slope Slow Down";
   "AL-Tunnel FW Stop Limit Slope" := "Slope Stop All";
   "AL-Tunnel FW Slow Limit Slope" := "Slope Slow Up";
   "AL-Up Stop Limit, Max Slope" := "Slope Stop Up";
   "AL-Down Stop Limit, Min Slope" := "Slope Stop Down";
END_REGION

REGION Network 4: Rotunda
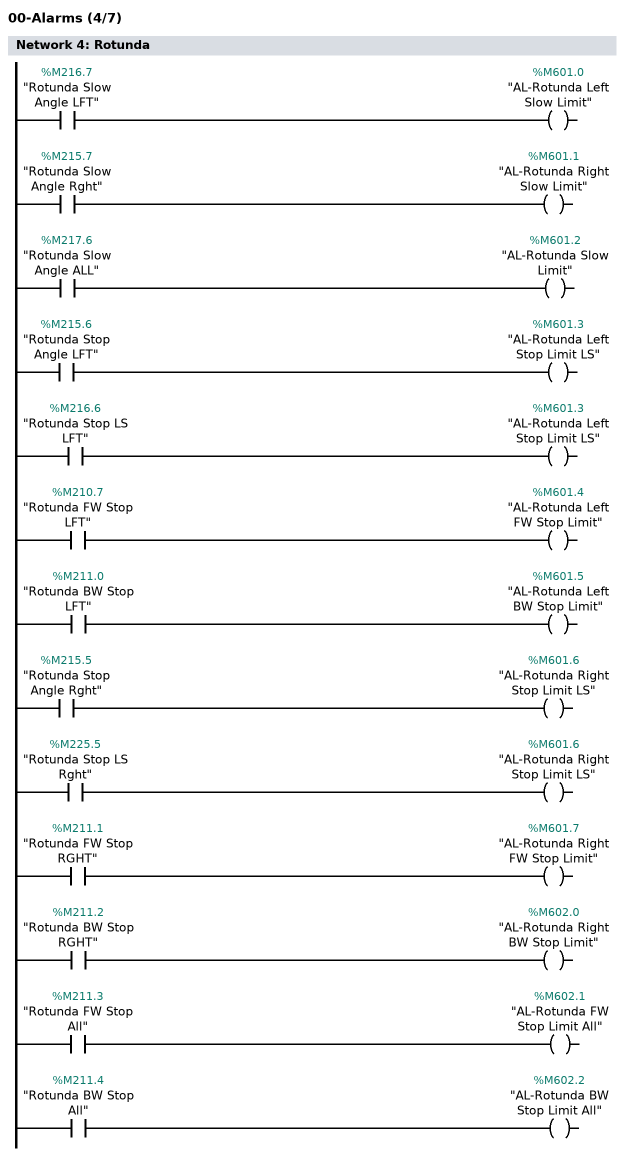
   RUNG wire#powerrail
      Contact( "Rotunda Slow Angle LFT" )
      Coil( "AL-Rotunda Left Slow Limit" )
   END_RUNG
   RUNG wire#powerrail
      Contact( "Rotunda Slow Angle Rght" )
      Coil( "AL-Rotunda Right Slow Limit" )
   END_RUNG
   RUNG wire#powerrail
      Contact( "Rotunda Slow Angle ALL" )
      Coil( "AL-Rotunda Slow Limit" )
   END_RUNG
   RUNG wire#powerrail
      Contact( "Rotunda Stop Angle LFT" )
      Coil( "AL-Rotunda Left Stop Limit LS" )
   END_RUNG
   RUNG wire#powerrail
      Contact( "Rotunda Stop LS LFT" )
      Coil( "AL-Rotunda Left Stop Limit LS" )
   END_RUNG
   RUNG wire#powerrail
      Contact( "Rotunda FW Stop LFT" )
      Coil( "AL-Rotunda Left FW Stop Limit" )
   END_RUNG
   RUNG wire#powerrail
      Contact( "Rotunda BW Stop LFT" )
      Coil( "AL-Rotunda Left BW Stop Limit" )
   END_RUNG
   RUNG wire#powerrail
      Contact( "Rotunda Stop Angle Rght" )
      Coil( "AL-Rotunda Right Stop Limit LS" )
   END_RUNG
   RUNG wire#powerrail
      Contact( "Rotunda Stop LS Rght" )
      Coil( "AL-Rotunda Right Stop Limit LS" )
   END_RUNG
   RUNG wire#powerrail
      Contact( "Rotunda FW Stop RGHT" )
      Coil( "AL-Rotunda Right FW Stop Limit" )
   END_RUNG
   RUNG wire#powerrail
      Contact( "Rotunda BW Stop RGHT" )
      Coil( "AL-Rotunda Right BW Stop Limit" )
   END_RUNG
   RUNG wire#powerrail
      Contact( "Rotunda FW Stop All" )
      Coil( "AL-Rotunda FW Stop Limit All" )
   END_RUNG
   RUNG wire#powerrail
      Contact( "Rotunda BW Stop All" )
      Coil( "AL-Rotunda BW Stop Limit All" )
   END_RUNG
   // the same network as SCL:
   "AL-Rotunda Left Slow Limit" := "Rotunda Slow Angle LFT";
   "AL-Rotunda Right Slow Limit" := "Rotunda Slow Angle Rght";
   "AL-Rotunda Slow Limit" := "Rotunda Slow Angle ALL";
   "AL-Rotunda Left Stop Limit LS" := "Rotunda Stop Angle LFT";
   "AL-Rotunda Left Stop Limit LS" := "Rotunda Stop LS LFT";
   "AL-Rotunda Left FW Stop Limit" := "Rotunda FW Stop LFT";
   "AL-Rotunda Left BW Stop Limit" := "Rotunda BW Stop LFT";
   "AL-Rotunda Right Stop Limit LS" := "Rotunda Stop Angle Rght";
   "AL-Rotunda Right Stop Limit LS" := "Rotunda Stop LS Rght";
   "AL-Rotunda Right FW Stop Limit" := "Rotunda FW Stop RGHT";
   "AL-Rotunda Right BW Stop Limit" := "Rotunda BW Stop RGHT";
   "AL-Rotunda FW Stop Limit All" := "Rotunda FW Stop All";
   "AL-Rotunda BW Stop Limit All" := "Rotunda BW Stop All";
END_REGION

REGION Network 5: Emergency
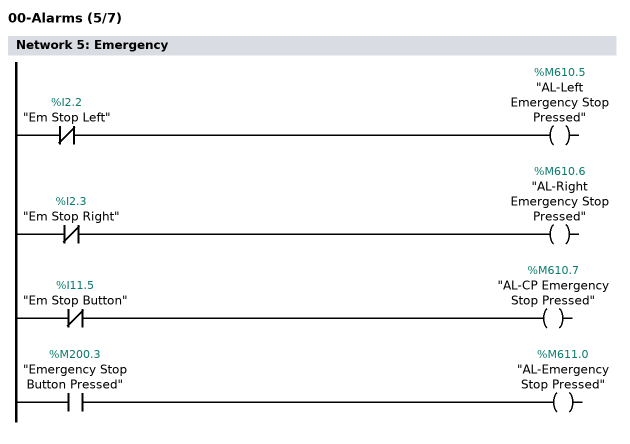
   RUNG wire#powerrail
      I_Contact( "Em Stop Left" )
      Coil( "AL-Left Emergency Stop Pressed" )
   END_RUNG
   RUNG wire#powerrail
      I_Contact( "Em Stop Right" )
      Coil( "AL-Right Emergency Stop Pressed" )
   END_RUNG
   RUNG wire#powerrail
      I_Contact( "Em Stop Button" )
      Coil( "AL-CP Emergency Stop Pressed" )
   END_RUNG
   RUNG wire#powerrail
      Contact( "Emergency Stop Button Pressed" )
      Coil( "AL-Emergency Stop Pressed" )
   END_RUNG
   // the same network as SCL:
   "AL-Left Emergency Stop Pressed" := NOT "Em Stop Left";
   "AL-Right Emergency Stop Pressed" := NOT "Em Stop Right";
   "AL-CP Emergency Stop Pressed" := NOT "Em Stop Button";
   "AL-Emergency Stop Pressed" := "Emergency Stop Button Pressed";
END_REGION

REGION Network 6: Cab
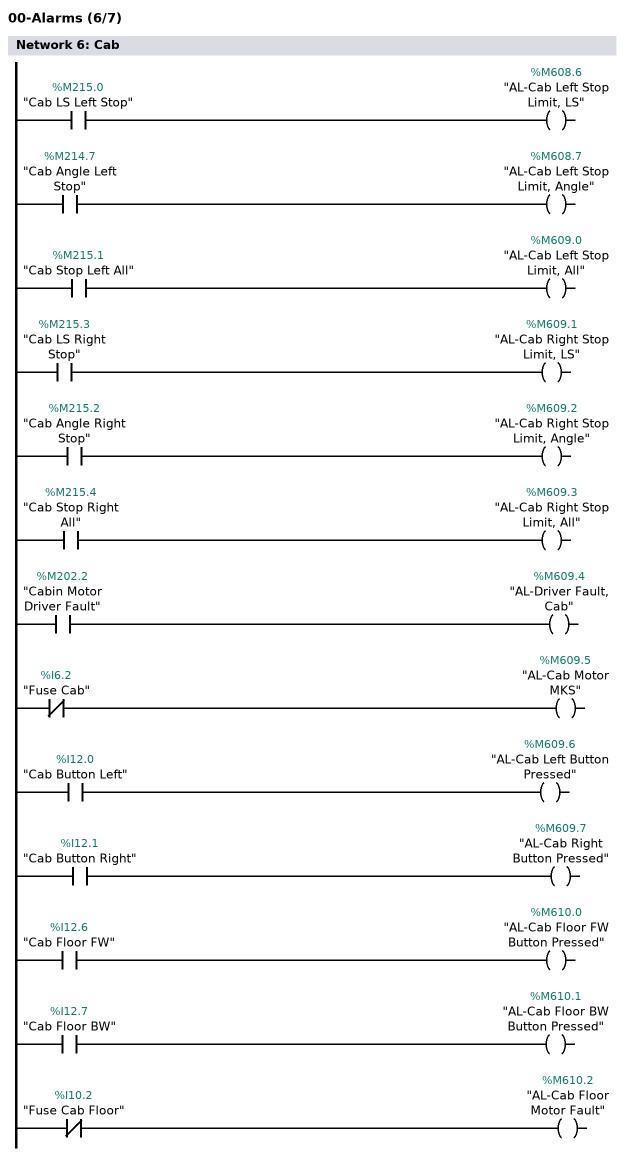
   RUNG wire#powerrail
      Contact( "Cab LS Left Stop" )
      Coil( "AL-Cab Left Stop Limit, LS" )
   END_RUNG
   RUNG wire#powerrail
      Contact( "Cab Angle Left Stop" )
      Coil( "AL-Cab Left Stop Limit, Angle" )
   END_RUNG
   RUNG wire#powerrail
      Contact( "Cab Stop Left All" )
      Coil( "AL-Cab Left Stop Limit, All" )
   END_RUNG
   RUNG wire#powerrail
      Contact( "Cab LS Right Stop" )
      Coil( "AL-Cab Right Stop Limit, LS" )
   END_RUNG
   RUNG wire#powerrail
      Contact( "Cab Angle Right Stop" )
      Coil( "AL-Cab Right Stop Limit, Angle" )
   END_RUNG
   RUNG wire#powerrail
      Contact( "Cab Stop Right All" )
      Coil( "AL-Cab Right Stop Limit, All" )
   END_RUNG
   RUNG wire#powerrail
      Contact( "Cabin Motor Driver Fault" )
      Coil( "AL-Driver Fault, Cab" )
   END_RUNG
   RUNG wire#powerrail
      I_Contact( "Fuse Cab" )
      Coil( "AL-Cab Motor MKS" )
   END_RUNG
   RUNG wire#powerrail
      Contact( "Cab Button Left" )
      Coil( "AL-Cab Left Button Pressed" )
   END_RUNG
   RUNG wire#powerrail
      Contact( "Cab Button Right" )
      Coil( "AL-Cab Right Button Pressed" )
   END_RUNG
   RUNG wire#powerrail
      Contact( "Cab Floor FW" )
      Coil( "AL-Cab Floor FW Button Pressed" )
   END_RUNG
   RUNG wire#powerrail
      Contact( "Cab Floor BW" )
      Coil( "AL-Cab Floor BW Button Pressed" )
   END_RUNG
   RUNG wire#powerrail
      I_Contact( "Fuse Cab Floor" )
      Coil( "AL-Cab Floor Motor Fault" )
   END_RUNG
   // the same network as SCL:
   "AL-Cab Left Stop Limit, LS" := "Cab LS Left Stop";
   "AL-Cab Left Stop Limit, Angle" := "Cab Angle Left Stop";
   "AL-Cab Left Stop Limit, All" := "Cab Stop Left All";
   "AL-Cab Right Stop Limit, LS" := "Cab LS Right Stop";
   "AL-Cab Right Stop Limit, Angle" := "Cab Angle Right Stop";
   "AL-Cab Right Stop Limit, All" := "Cab Stop Right All";
   "AL-Driver Fault, Cab" := "Cabin Motor Driver Fault";
   "AL-Cab Motor MKS" := NOT "Fuse Cab";
   "AL-Cab Left Button Pressed" := "Cab Button Left";
   "AL-Cab Right Button Pressed" := "Cab Button Right";
   "AL-Cab Floor FW Button Pressed" := "Cab Floor FW";
   "AL-Cab Floor BW Button Pressed" := "Cab Floor BW";
   "AL-Cab Floor Motor Fault" := NOT "Fuse Cab Floor";
END_REGION

REGION Network 7: Canopy
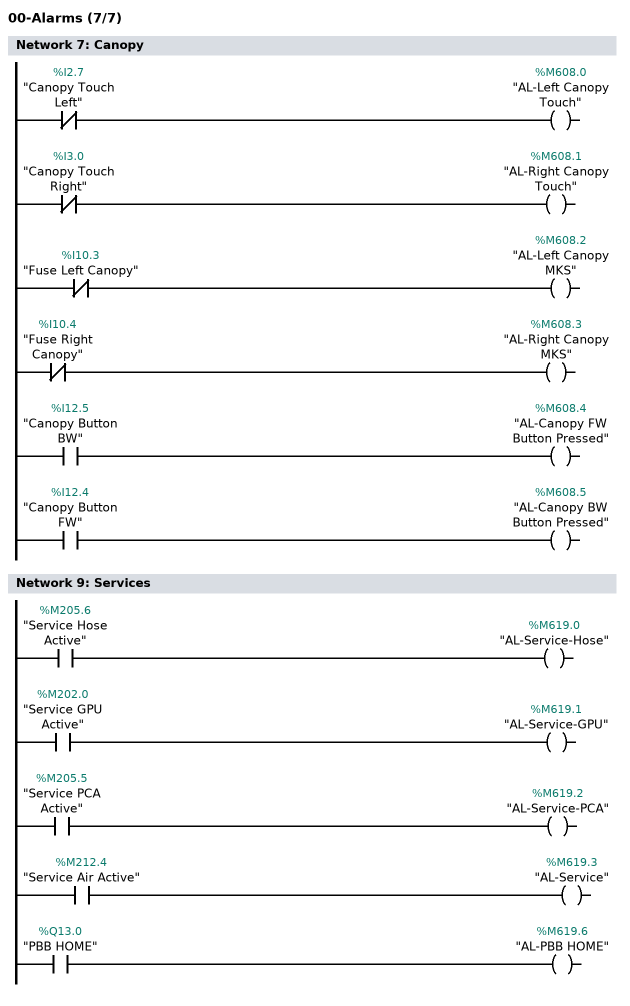
   RUNG wire#powerrail
      I_Contact( "Canopy Touch Left" )
      Coil( "AL-Left Canopy Touch" )
   END_RUNG
   RUNG wire#powerrail
      I_Contact( "Canopy Touch Right" )
      Coil( "AL-Right Canopy Touch" )
   END_RUNG
   RUNG wire#powerrail
      I_Contact( "Fuse Left Canopy" )
      Coil( "AL-Left Canopy MKS" )
   END_RUNG
   RUNG wire#powerrail
      I_Contact( "Fuse Right Canopy" )
      Coil( "AL-Right Canopy MKS" )
   END_RUNG
   RUNG wire#powerrail
      Contact( "Canopy Button BW" )
      Coil( "AL-Canopy FW Button Pressed" )
   END_RUNG
   RUNG wire#powerrail
      Contact( "Canopy Button FW" )
      Coil( "AL-Canopy BW Button Pressed" )
   END_RUNG
   // the same network as SCL:
   "AL-Left Canopy Touch" := NOT "Canopy Touch Left";
   "AL-Right Canopy Touch" := NOT "Canopy Touch Right";
   "AL-Left Canopy MKS" := NOT "Fuse Left Canopy";
   "AL-Right Canopy MKS" := NOT "Fuse Right Canopy";
   "AL-Canopy FW Button Pressed" := "Canopy Button BW";
   "AL-Canopy BW Button Pressed" := "Canopy Button FW";
END_REGION

REGION Network 8: PCA and GPU Service
END_REGION

REGION Network 9: Services
   RUNG wire#powerrail
      Contact( "Service Hose Active" )
      Coil( "AL-Service-Hose" )
   END_RUNG
   RUNG wire#powerrail
      Contact( "Service GPU Active" )
      Coil( "AL-Service-GPU" )
   END_RUNG
   RUNG wire#powerrail
      Contact( "Service PCA Active" )
      Coil( "AL-Service-PCA" )
   END_RUNG
   RUNG wire#powerrail
      Contact( "Service Air Active" )
      Coil( "AL-Service" )
   END_RUNG
   RUNG wire#powerrail
      Contact( "PBB HOME" )
      Coil( "AL-PBB HOME" )
   END_RUNG
   // the same network as SCL:
   "AL-Service-Hose" := "Service Hose Active";
   "AL-Service-GPU" := "Service GPU Active";
   "AL-Service-PCA" := "Service PCA Active";
   "AL-Service" := "Service Air Active";
   "AL-PBB HOME" := "PBB HOME";
END_REGION
END_ORGANIZATION_BLOCK

ORGANIZATION_BLOCK "11-Bridge Movements"   // OB123, LAD, ProgramCycle
TITLE = Wheel
{ S7_Optimized_Access := 'TRUE' }
VERSION : 0.1
// stored: AutoNumber true, IsIECCheckEnabled false, SetENOAutomatically false
   VAR_INPUT
      Initial_Call : Bool;   // Initial call of this OB
      Remanence : Bool;   // =True, if remanent data are available
   END_VAR
   VAR_TEMP   // added for the SCL form of the ladder/FBD networks
      _w1 : Bool;
      _w2 : Bool;
      _w3 : Bool;
      _w4 : Bool;
   END_VAR
BEGIN

REGION Network 1: JoyStick MID
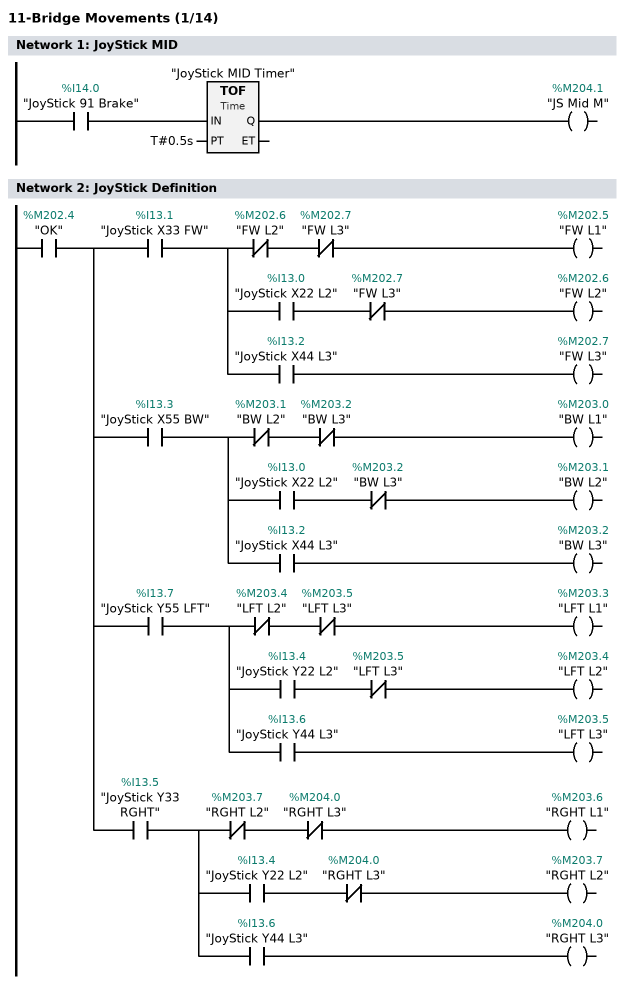
   RUNG wire#powerrail
      Contact( "JoyStick 91 Brake" )
      { S7_Templates := "time_type := Time" } "JoyStick MID Timer".TOF(pt := T#0.5s, et =>)
      Coil( "JS Mid M" )
   END_RUNG
   // the same network as SCL:
   "JoyStick MID Timer".TOF(IN := "JoyStick 91 Brake", PT := T#0.5s);
   "JS Mid M" := "JoyStick MID Timer".Q;
END_REGION

REGION Network 2: JoyStick Definition
   RUNG wire#powerrail
      Contact( "OK" )
      wire#w1
      Contact( "JoyStick X33 FW" )
      wire#w2
      I_Contact( "FW L2" )
      I_Contact( "FW L3" )
      Coil( "FW L1" )
   END_RUNG
   RUNG wire#w2
      Contact( "JoyStick X22 L2" )
      I_Contact( "FW L3" )
      Coil( "FW L2" )
   END_RUNG
   RUNG wire#w2
      Contact( "JoyStick X44 L3" )
      Coil( "FW L3" )
   END_RUNG
   RUNG wire#w1
      Contact( "JoyStick X55 BW" )
      wire#w3
      I_Contact( "BW L2" )
      I_Contact( "BW L3" )
      Coil( "BW L1" )
   END_RUNG
   RUNG wire#w3
      Contact( "JoyStick X22 L2" )
      I_Contact( "BW L3" )
      Coil( "BW L2" )
   END_RUNG
   RUNG wire#w3
      Contact( "JoyStick X44 L3" )
      Coil( "BW L3" )
   END_RUNG
   RUNG wire#w1
      Contact( "JoyStick Y55 LFT" )
      wire#w4
      I_Contact( "LFT L2" )
      I_Contact( "LFT L3" )
      Coil( "LFT L1" )
   END_RUNG
   RUNG wire#w4
      Contact( "JoyStick Y22 L2" )
      I_Contact( "LFT L3" )
      Coil( "LFT L2" )
   END_RUNG
   RUNG wire#w4
      Contact( "JoyStick Y44 L3" )
      Coil( "LFT L3" )
   END_RUNG
   RUNG wire#w1
      Contact( "JoyStick Y33 RGHT" )
      wire#w5
      I_Contact( "RGHT L2" )
      I_Contact( "RGHT L3" )
      Coil( "RGHT L1" )
   END_RUNG
   RUNG wire#w5
      Contact( "JoyStick Y22 L2" )
      I_Contact( "RGHT L3" )
      Coil( "RGHT L2" )
   END_RUNG
   RUNG wire#w5
      Contact( "JoyStick Y44 L3" )
      Coil( "RGHT L3" )
   END_RUNG
   // the same network as SCL:
   #_w1 := "OK" AND "JoyStick X33 FW";
   "FW L1" := #_w1 AND NOT "FW L2" AND NOT "FW L3";
   "FW L2" := #_w1 AND "JoyStick X22 L2" AND NOT "FW L3";
   "FW L3" := #_w1 AND "JoyStick X44 L3";
   #_w2 := "OK" AND "JoyStick X55 BW";
   "BW L1" := #_w2 AND NOT "BW L2" AND NOT "BW L3";
   "BW L2" := #_w2 AND "JoyStick X22 L2" AND NOT "BW L3";
   "BW L3" := #_w2 AND "JoyStick X44 L3";
   #_w3 := "OK" AND "JoyStick Y55 LFT";
   "LFT L1" := #_w3 AND NOT "LFT L2" AND NOT "LFT L3";
   "LFT L2" := #_w3 AND "JoyStick Y22 L2" AND NOT "LFT L3";
   "LFT L3" := #_w3 AND "JoyStick Y44 L3";
   #_w4 := "OK" AND "JoyStick Y33 RGHT";
   "RGHT L1" := #_w4 AND NOT "RGHT L2" AND NOT "RGHT L3";
   "RGHT L2" := #_w4 AND "JoyStick Y22 L2" AND NOT "RGHT L3";
   "RGHT L3" := #_w4 AND "JoyStick Y44 L3";
END_REGION

REGION Network 3: JoyStick Cross Definition
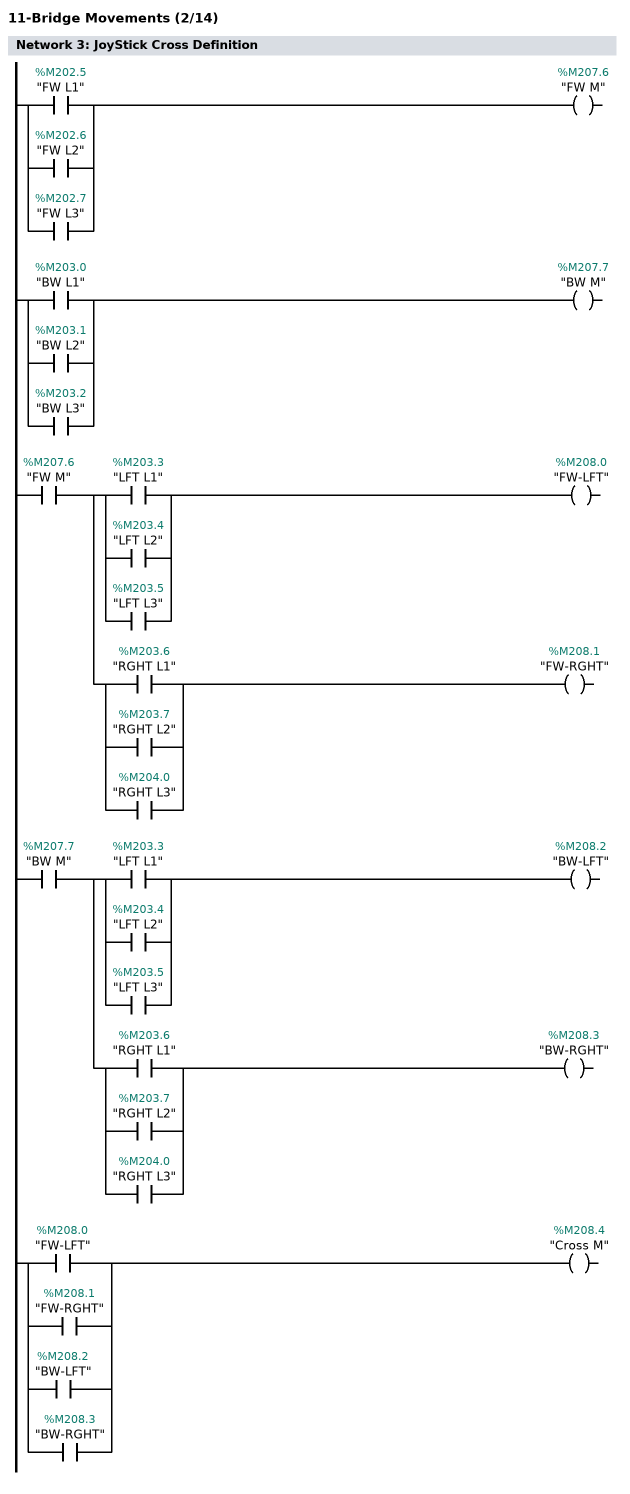
   RUNG wire#powerrail
      Contact( "FW L1" )
      wire#w1
      Coil( "FW M" )
   END_RUNG
   RUNG wire#powerrail
      Contact( "FW L2" )
   END_RUNG wire#w1
   RUNG wire#powerrail
      Contact( "FW L3" )
   END_RUNG wire#w1
   RUNG wire#powerrail
      Contact( "BW L1" )
      wire#w2
      Coil( "BW M" )
   END_RUNG
   RUNG wire#powerrail
      Contact( "BW L2" )
   END_RUNG wire#w2
   RUNG wire#powerrail
      Contact( "BW L3" )
   END_RUNG wire#w2
   RUNG wire#powerrail
      Contact( "FW M" )
      wire#w3
      Contact( "LFT L1" )
      wire#w4
      Coil( "FW-LFT" )
   END_RUNG
   RUNG wire#w3
      Contact( "LFT L2" )
   END_RUNG wire#w4
   RUNG wire#w3
      Contact( "LFT L3" )
   END_RUNG wire#w4
   RUNG wire#w3
      Contact( "RGHT L1" )
      wire#w5
      Coil( "FW-RGHT" )
   END_RUNG
   RUNG wire#w3
      Contact( "RGHT L2" )
   END_RUNG wire#w5
   RUNG wire#w3
      Contact( "RGHT L3" )
   END_RUNG wire#w5
   RUNG wire#powerrail
      Contact( "BW M" )
      wire#w6
      Contact( "LFT L1" )
      wire#w7
      Coil( "BW-LFT" )
   END_RUNG
   RUNG wire#w6
      Contact( "LFT L2" )
   END_RUNG wire#w7
   RUNG wire#w6
      Contact( "LFT L3" )
   END_RUNG wire#w7
   RUNG wire#w6
      Contact( "RGHT L1" )
      wire#w8
      Coil( "BW-RGHT" )
   END_RUNG
   RUNG wire#w6
      Contact( "RGHT L2" )
   END_RUNG wire#w8
   RUNG wire#w6
      Contact( "RGHT L3" )
   END_RUNG wire#w8
   RUNG wire#powerrail
      Contact( "FW-LFT" )
      wire#w9
      Coil( "Cross M" )
   END_RUNG
   RUNG wire#powerrail
      Contact( "FW-RGHT" )
   END_RUNG wire#w9
   RUNG wire#powerrail
      Contact( "BW-LFT" )
   END_RUNG wire#w9
   RUNG wire#powerrail
      Contact( "BW-RGHT" )
   END_RUNG wire#w9
   // the same network as SCL:
   "FW M" := "FW L1" OR "FW L2" OR "FW L3";
   "BW M" := "BW L1" OR "BW L2" OR "BW L3";
   "FW-LFT" := "FW M" AND ("LFT L1" OR "LFT L2" OR "LFT L3");
   "FW-RGHT" := "FW M" AND ("RGHT L1" OR "RGHT L2" OR "RGHT L3");
   "BW-LFT" := "BW M" AND ("LFT L1" OR "LFT L2" OR "LFT L3");
   "BW-RGHT" := "BW M" AND ("RGHT L1" OR "RGHT L2" OR "RGHT L3");
   "Cross M" := "FW-LFT" OR "FW-RGHT" OR "BW-LFT" OR "BW-RGHT";
END_REGION

REGION Network 4: Speed Settings
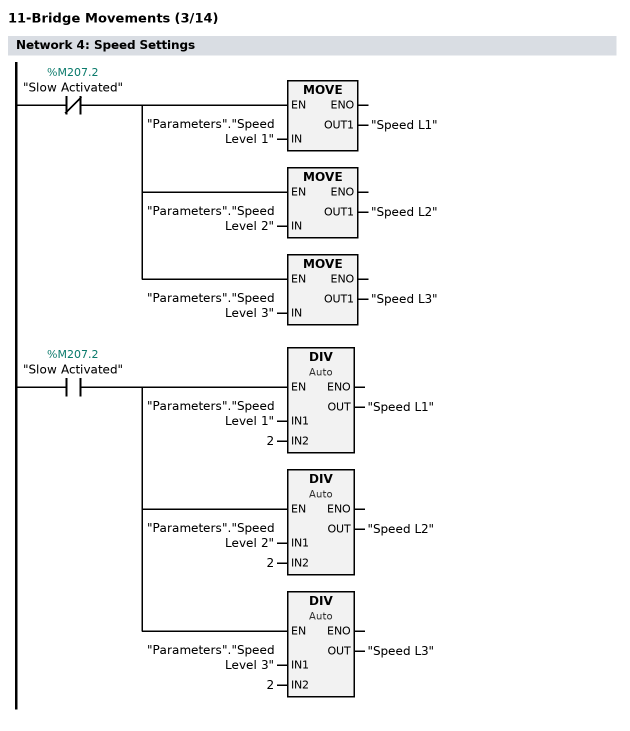
   RUNG wire#powerrail
      I_Contact( "Slow Activated" )
      wire#w1
      Move(in := "Parameters"."Speed Level 1", out1 => "Speed L1")
   END_RUNG
   RUNG wire#w1
      Move(in := "Parameters"."Speed Level 2", out1 => "Speed L2")
   END_RUNG
   RUNG wire#w1
      Move(in := "Parameters"."Speed Level 3", out1 => "Speed L3")
   END_RUNG
   RUNG wire#powerrail
      Contact( "Slow Activated" )
      wire#w2
      Div(in1 := "Parameters"."Speed Level 1", in2 := 2, out => "Speed L1")
   END_RUNG
   RUNG wire#w2
      Div(in1 := "Parameters"."Speed Level 2", in2 := 2, out => "Speed L2")
   END_RUNG
   RUNG wire#w2
      Div(in1 := "Parameters"."Speed Level 3", in2 := 2, out => "Speed L3")
   END_RUNG
   // the same network as SCL:
   IF NOT "Slow Activated" THEN
       "Speed L1" := "Parameters"."Speed Level 1";
       "Speed L2" := "Parameters"."Speed Level 2";
       "Speed L3" := "Parameters"."Speed Level 3";
   END_IF;
   IF "Slow Activated" THEN
       "Speed L1" := "Parameters"."Speed Level 1" / 2;
       "Speed L2" := "Parameters"."Speed Level 2" / 2;
       "Speed L3" := "Parameters"."Speed Level 3" / 2;
   END_IF;
END_REGION

REGION Network 5: Speed Definition
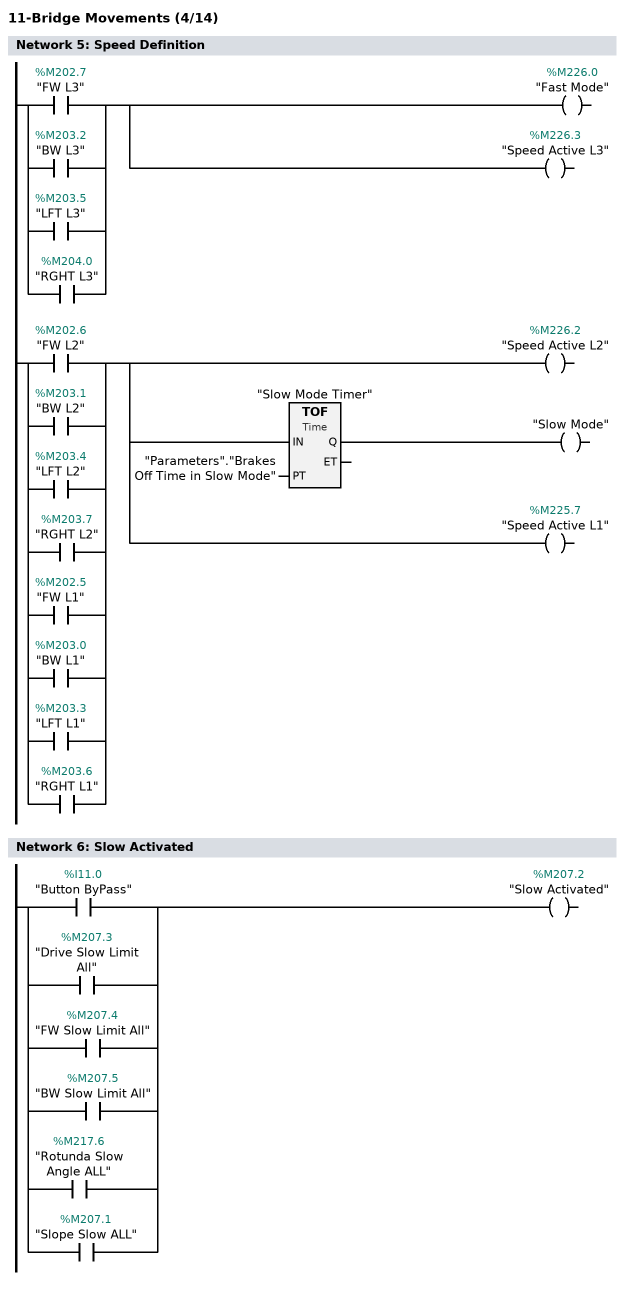
   RUNG wire#powerrail
      Contact( "FW L3" )
      wire#w1
      Coil( "Fast Mode" )
   END_RUNG
   RUNG wire#powerrail
      Contact( "BW L3" )
   END_RUNG wire#w1
   RUNG wire#powerrail
      Contact( "LFT L3" )
   END_RUNG wire#w1
   RUNG wire#powerrail
      Contact( "RGHT L3" )
   END_RUNG wire#w1
   RUNG wire#w1
      Coil( "Speed Active L3" )
   END_RUNG
   RUNG wire#powerrail
      Contact( "FW L2" )
      wire#w2
      Coil( "Speed Active L2" )
   END_RUNG
   RUNG wire#powerrail
      Contact( "BW L2" )
   END_RUNG wire#w2
   RUNG wire#powerrail
      Contact( "LFT L2" )
   END_RUNG wire#w2
   RUNG wire#powerrail
      Contact( "RGHT L2" )
   END_RUNG wire#w2
   RUNG wire#powerrail
      Contact( "FW L1" )
   END_RUNG wire#w2
   RUNG wire#powerrail
      Contact( "BW L1" )
   END_RUNG wire#w2
   RUNG wire#powerrail
      Contact( "LFT L1" )
   END_RUNG wire#w2
   RUNG wire#powerrail
      Contact( "RGHT L1" )
   END_RUNG wire#w2
   RUNG wire#w2
      { S7_Templates := "time_type := Time" } "Slow Mode Timer".TOF(pt := "Parameters"."Brakes Off Time in Slow Mode", et =>)
      Coil( "Slow Mode" )
   END_RUNG
   RUNG wire#w2
      Coil( "Speed Active L1" )
   END_RUNG
   // the same network as SCL:
   "Fast Mode" := "FW L3" OR "BW L3" OR "LFT L3" OR "RGHT L3";
   "Speed Active L3" := "Fast Mode";
   "Speed Active L2" := "FW L2" OR "BW L2" OR "LFT L2" OR "RGHT L2" OR "FW L1" OR "BW L1" OR "LFT L1" OR "RGHT L1";
   "Slow Mode Timer".TOF(IN := "Speed Active L2", PT := "Parameters"."Brakes Off Time in Slow Mode");
   "Slow Mode" := "Slow Mode Timer".Q;
   "Speed Active L1" := "Speed Active L2";
END_REGION

REGION Network 6: Slow Activated
   RUNG wire#powerrail
      Contact( "Button ByPass" )
      wire#w1
      Coil( "Slow Activated" )
   END_RUNG
   RUNG wire#powerrail
      Contact( "Drive Slow Limit All" )
   END_RUNG wire#w1
   RUNG wire#powerrail
      Contact( "FW Slow Limit All" )
   END_RUNG wire#w1
   RUNG wire#powerrail
      Contact( "BW Slow Limit All" )
   END_RUNG wire#w1
   RUNG wire#powerrail
      Contact( "Rotunda Slow Angle ALL" )
   END_RUNG wire#w1
   RUNG wire#powerrail
      Contact( "Slope Slow ALL" )
   END_RUNG wire#w1
   // the same network as SCL:
   "Slow Activated" := "Button ByPass" OR "Drive Slow Limit All" OR "FW Slow Limit All" OR "BW Slow Limit All" OR "Rotunda Slow Angle ALL" OR "Slope Slow ALL";
END_REGION

REGION Network 7: Tunnel FW Slow Limits
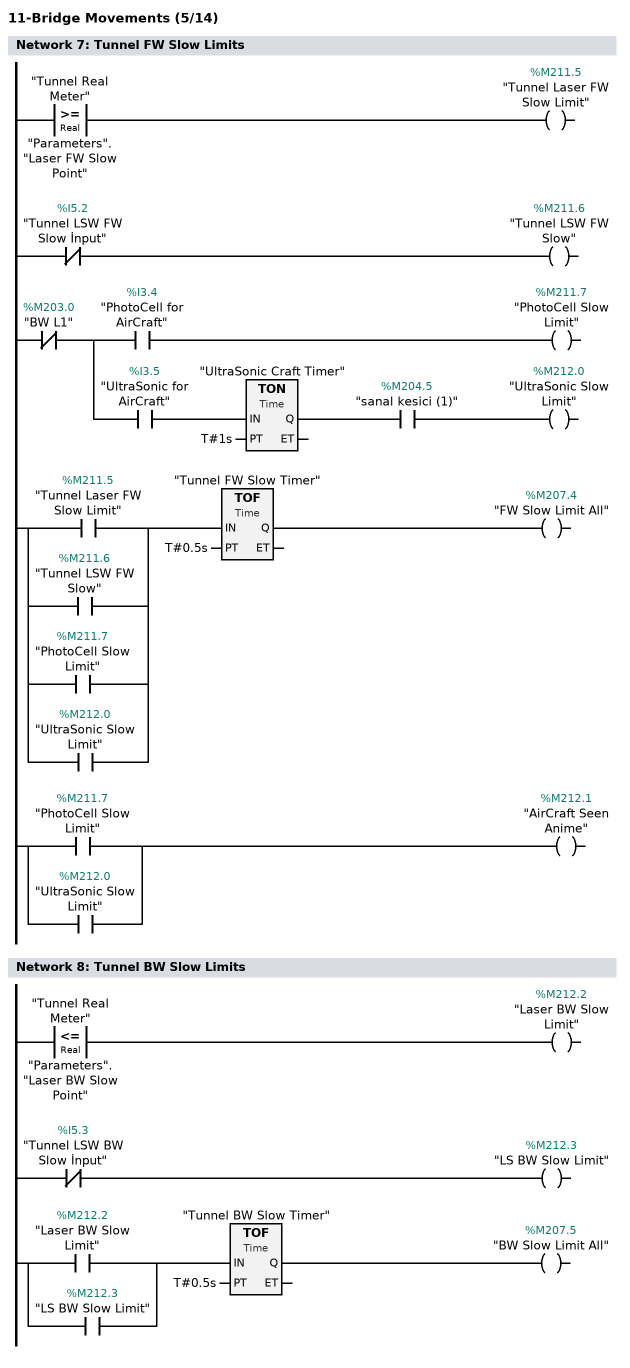
   RUNG wire#powerrail
      { S7_Templates := "SrcType := Real" } GE_Contact(in1 := "Tunnel Real Meter", in2 := "Parameters"."Laser FW Slow Point")
      Coil( "Tunnel Laser FW Slow Limit" )
   END_RUNG
   RUNG wire#powerrail
      I_Contact( "Tunnel LSW FW Slow İnput" )
      Coil( "Tunnel LSW FW Slow" )
   END_RUNG
   RUNG wire#powerrail
      I_Contact( "BW L1" )
      wire#w1
      Contact( "PhotoCell for AirCraft" )
      Coil( "PhotoCell Slow Limit" )
   END_RUNG
   RUNG wire#w1
      Contact( "UltraSonic for AirCraft" )
      { S7_Templates := "time_type := Time" } "UltraSonic Craft Timer".TON(pt := T#1s, et =>)
      Contact( "sanal kesici (1)" )
      Coil( "UltraSonic Slow Limit" )
   END_RUNG
   RUNG wire#powerrail
      Contact( "Tunnel Laser FW Slow Limit" )
      wire#w2
      { S7_Templates := "time_type := Time" } "Tunnel FW Slow Timer".TOF(pt := T#0.5s, et =>)
      Coil( "FW Slow Limit All" )
   END_RUNG
   RUNG wire#powerrail
      Contact( "Tunnel LSW FW Slow" )
   END_RUNG wire#w2
   RUNG wire#powerrail
      Contact( "PhotoCell Slow Limit" )
   END_RUNG wire#w2
   RUNG wire#powerrail
      Contact( "UltraSonic Slow Limit" )
   END_RUNG wire#w2
   RUNG wire#powerrail
      Contact( "PhotoCell Slow Limit" )
      wire#w3
      Coil( "AirCraft Seen Anime" )
   END_RUNG
   RUNG wire#powerrail
      Contact( "UltraSonic Slow Limit" )
   END_RUNG wire#w3
   // the same network as SCL:
   "Tunnel Laser FW Slow Limit" := "Tunnel Real Meter" >= "Parameters"."Laser FW Slow Point";
   "Tunnel LSW FW Slow" := NOT "Tunnel LSW FW Slow İnput";
   "PhotoCell Slow Limit" := NOT "BW L1" AND "PhotoCell for AirCraft";
   "UltraSonic Craft Timer".TON(IN := NOT "BW L1" AND "UltraSonic for AirCraft", PT := T#1s);
   "UltraSonic Slow Limit" := "UltraSonic Craft Timer".Q AND "sanal kesici (1)";
   "Tunnel FW Slow Timer".TOF(IN := "Tunnel Laser FW Slow Limit" OR "Tunnel LSW FW Slow" OR "PhotoCell Slow Limit" OR "UltraSonic Slow Limit",
                           PT := T#0.5s);
   "FW Slow Limit All" := "Tunnel FW Slow Timer".Q;
   "AirCraft Seen Anime" := "PhotoCell Slow Limit" OR "UltraSonic Slow Limit";
END_REGION

REGION Network 8: Tunnel BW Slow Limits
   RUNG wire#powerrail
      { S7_Templates := "SrcType := Real" } LE_Contact(in1 := "Tunnel Real Meter", in2 := "Parameters"."Laser BW Slow Point")
      Coil( "Laser BW Slow Limit" )
   END_RUNG
   RUNG wire#powerrail
      I_Contact( "Tunnel LSW BW Slow İnput" )
      Coil( "LS BW Slow Limit" )
   END_RUNG
   RUNG wire#powerrail
      Contact( "Laser BW Slow Limit" )
      wire#w1
      { S7_Templates := "time_type := Time" } "Tunnel BW Slow Timer".TOF(pt := T#0.5s, et =>)
      Coil( "BW Slow Limit All" )
   END_RUNG
   RUNG wire#powerrail
      Contact( "LS BW Slow Limit" )
   END_RUNG wire#w1
   // the same network as SCL:
   "Laser BW Slow Limit" := "Tunnel Real Meter" <= "Parameters"."Laser BW Slow Point";
   "LS BW Slow Limit" := NOT "Tunnel LSW BW Slow İnput";
   "Tunnel BW Slow Timer".TOF(IN := "Laser BW Slow Limit" OR "LS BW Slow Limit", PT := T#0.5s);
   "BW Slow Limit All" := "Tunnel BW Slow Timer".Q;
END_REGION

REGION Network 9: Tunnel FW Stop Limits
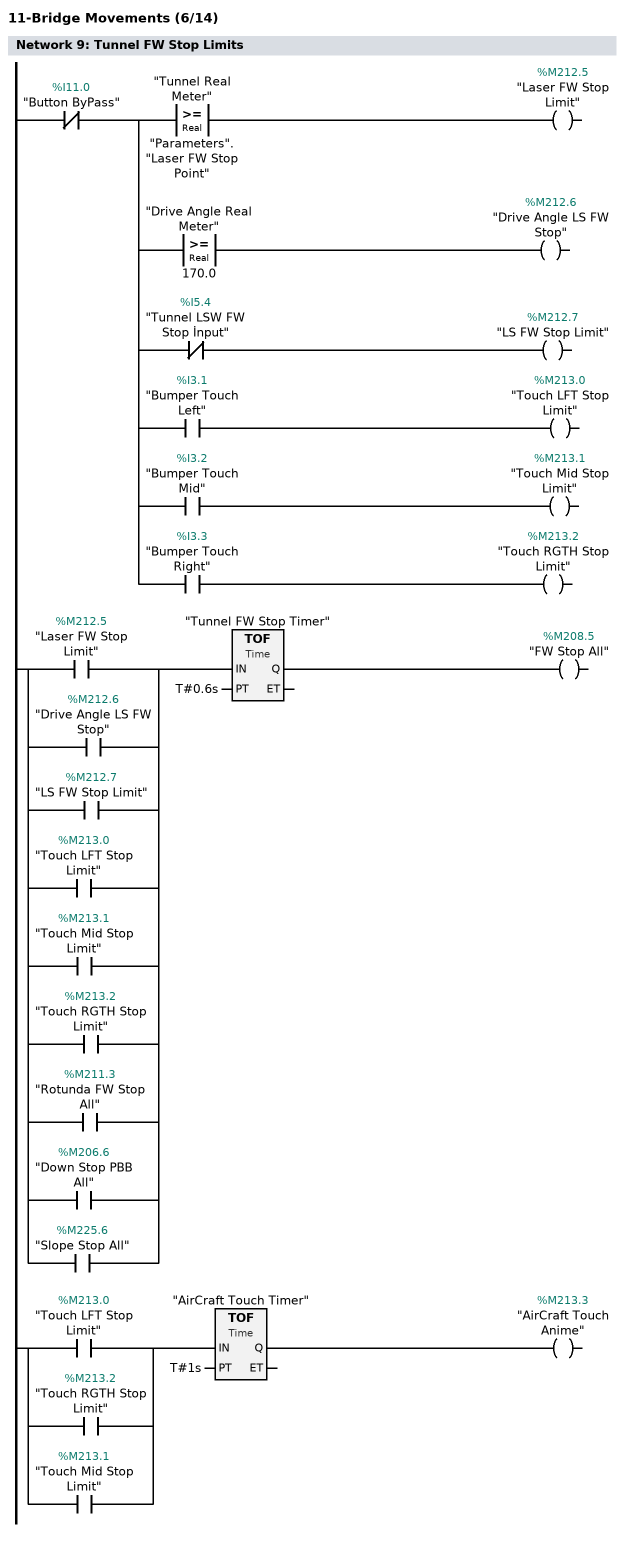
   RUNG wire#powerrail
      I_Contact( "Button ByPass" )
      wire#w1
      { S7_Templates := "SrcType := Real" } GE_Contact(in1 := "Tunnel Real Meter", in2 := "Parameters"."Laser FW Stop Point")
      Coil( "Laser FW Stop Limit" )
   END_RUNG
   RUNG wire#w1
      { S7_Templates := "SrcType := Real" } GE_Contact(in1 := "Drive Angle Real Meter", in2 := 170.0)
      Coil( "Drive Angle LS FW Stop" )
   END_RUNG
   RUNG wire#w1
      I_Contact( "Tunnel LSW FW Stop İnput" )
      Coil( "LS FW Stop Limit" )
   END_RUNG
   RUNG wire#w1
      Contact( "Bumper Touch Left" )
      Coil( "Touch LFT Stop Limit" )
   END_RUNG
   RUNG wire#w1
      Contact( "Bumper Touch Mid" )
      Coil( "Touch Mid Stop Limit" )
   END_RUNG
   RUNG wire#w1
      Contact( "Bumper Touch Right" )
      Coil( "Touch RGTH Stop Limit" )
   END_RUNG
   RUNG wire#powerrail
      Contact( "Laser FW Stop Limit" )
      wire#w2
      { S7_Templates := "time_type := Time" } "Tunnel FW Stop Timer".TOF(pt := T#0.6s, et =>)
      Coil( "FW Stop All" )
   END_RUNG
   RUNG wire#powerrail
      Contact( "Drive Angle LS FW Stop" )
   END_RUNG wire#w2
   RUNG wire#powerrail
      Contact( "LS FW Stop Limit" )
   END_RUNG wire#w2
   RUNG wire#powerrail
      Contact( "Touch LFT Stop Limit" )
   END_RUNG wire#w2
   RUNG wire#powerrail
      Contact( "Touch Mid Stop Limit" )
   END_RUNG wire#w2
   RUNG wire#powerrail
      Contact( "Touch RGTH Stop Limit" )
   END_RUNG wire#w2
   RUNG wire#powerrail
      Contact( "Rotunda FW Stop All" )
   END_RUNG wire#w2
   RUNG wire#powerrail
      Contact( "Down Stop PBB All" )
   END_RUNG wire#w2
   RUNG wire#powerrail
      Contact( "Slope Stop All" )
   END_RUNG wire#w2
   RUNG wire#powerrail
      Contact( "Touch LFT Stop Limit" )
      wire#w3
      { S7_Templates := "time_type := Time" } "AirCraft Touch Timer".TOF(pt := T#1s, et =>)
      Coil( "AirCraft Touch Anime" )
   END_RUNG
   RUNG wire#powerrail
      Contact( "Touch RGTH Stop Limit" )
   END_RUNG wire#w3
   RUNG wire#powerrail
      Contact( "Touch Mid Stop Limit" )
   END_RUNG wire#w3
   // the same network as SCL:
   "Laser FW Stop Limit" := NOT "Button ByPass" AND ("Tunnel Real Meter" >= "Parameters"."Laser FW Stop Point");
   "Drive Angle LS FW Stop" := NOT "Button ByPass" AND ("Drive Angle Real Meter" >= 170.0);
   "LS FW Stop Limit" := NOT "Button ByPass" AND NOT "Tunnel LSW FW Stop İnput";
   "Touch LFT Stop Limit" := NOT "Button ByPass" AND "Bumper Touch Left";
   "Touch Mid Stop Limit" := NOT "Button ByPass" AND "Bumper Touch Mid";
   "Touch RGTH Stop Limit" := NOT "Button ByPass" AND "Bumper Touch Right";
   "Tunnel FW Stop Timer".TOF(IN := "Laser FW Stop Limit" OR "Drive Angle LS FW Stop" OR "LS FW Stop Limit" OR "Touch LFT Stop Limit" OR "Touch Mid Stop Limit" OR "Touch RGTH Stop Limit" OR "Rotunda FW Stop All" OR "Down Stop PBB All" OR "Slope Stop All",
                           PT := T#0.6s);
   "FW Stop All" := "Tunnel FW Stop Timer".Q;
   "AirCraft Touch Timer".TOF(IN := "Touch LFT Stop Limit" OR "Touch RGTH Stop Limit" OR "Touch Mid Stop Limit",
                           PT := T#1s);
   "AirCraft Touch Anime" := "AirCraft Touch Timer".Q;
END_REGION

REGION Network 10: Tunnel BW Stop Limits
